(* IEC 61131-3 sources: horner-cscape-mcp/fixtures/st_library, 17 files *)

(* ---- analog_scaling_bounds.st ---- *)
(* ============================================================================
 * Title:       FB_AnalogScalingOutOfBounds
 * Description: Industrial Analog Scaling with Out-of-Bounds & Sensor Diagnostics.
 * Features:
 *   - Linear interpolation: Raw ADC / mA counts to Engineering Units (EU)
 *   - Out-of-bounds detection: 4-20mA open-loop wire-break and short-circuit faults
 *   - Configurable exponential smoothing digital filter for noisy plant signals
 *   - Output clamping to user process limits
 *   - Fail-safe fallback strategies (Hold Last Valid or Drive to Safe Preset)
 *   - Real-time sensor quality status and latched diagnostic error codes
 * Language:    IEC 61131-3 Structured Text (Pure ST)
 * ============================================================================ *)

FUNCTION_BLOCK FB_AnalogScalingOutOfBounds
VAR_INPUT
    RawIn : REAL := 0.0;                  (* Unscaled raw analog reading from ADC / PLC input *)
    RawMin : REAL := 4000.0;              (* Raw value corresponding to 0% range (e.g. 4.00 mA = 4000) *)
    RawMax : REAL := 20000.0;             (* Raw value corresponding to 100% range (e.g. 20.00 mA = 20000) *)
    EngMin : REAL := 0.0;                 (* Engineering units minimum (e.g. 0.0 Bar, Deg C, or RPM) *)
    EngMax : REAL := 100.0;               (* Engineering units maximum (e.g. 100.0 Bar, Deg C, or RPM) *)
    UnderflowTolerance : REAL := 400.0;   (* Margin below RawMin before declaring wire break (e.g. < 3.6 mA) *)
    OverflowTolerance : REAL := 800.0;    (* Margin above RawMax before declaring short circuit (e.g. > 20.8 mA) *)
    ClampOutput : BOOL := TRUE;           (* TRUE = constrain output between EngMin and EngMax *)
    FilterAlpha : REAL := 0.20;           (* Digital 1st-order filter factor (0.01 = heavy, 1.0 = bypass) *)
    FailSafeMode : INT := 0;              (* Fallback action on fault: 0 = Preset SafeValue, 1 = Hold Last Valid *)
    FailSafeValue : REAL := 0.0;          (* Fallback value emitted when FailSafeMode = 0 during fault *)
    ResetFault : BOOL := FALSE;           (* Pushbutton input to reset latched fault flags *)
END_VAR

VAR_OUTPUT
    ScaledValue : REAL := 0.0;            (* Final conditioned engineering units value *)
    RawFiltered : REAL := 0.0;            (* Filtered raw analog signal before scaling *)
    QualityOK : BOOL := TRUE;             (* Sensor signal is healthy and within legal electrical bounds *)
    AlarmUnderflow : BOOL := FALSE;       (* Active wire-break / open-loop / disconnected transmitter *)
    AlarmOverflow : BOOL := FALSE;        (* Active over-current / wiring short / ADC saturation *)
    LatchedFault : BOOL := FALSE;         (* Latch indicating an abnormal electrical event occurred *)
    ErrorCode : INT := 0;                 (* Diagnostics: 0=OK, 1=Underflow/Break, 2=Overflow/Short, 3=Config *)
END_VAR

VAR
    RawSpan : REAL := 16000.0;            (* Calculated raw range (RawMax - RawMin) *)
    EngSpan : REAL := 100.0;              (* Calculated engineering range (EngMax - EngMin) *)
    NormalizedFrac : REAL := 0.0;         (* Fraction between 0.0 and 1.0 *)
    CalculatedEng : REAL := 0.0;          (* Scaled value before clamping *)
    LastValidValue : REAL := 0.0;         (* Memory storing last known healthy measurement *)
    FilterInitialized : BOOL := FALSE;    (* Flag for initializing filter on first scan *)
END_VAR

(* 1. Reset Diagnostic Faults *)
IF ResetFault THEN
    LatchedFault := FALSE;
    ErrorCode := 0;
END_IF;

(* 2. Configuration Validation *)
RawSpan := RawMax - RawMin;
EngSpan := EngMax - EngMin;

IF ABS(RawSpan) < 0.001 THEN
    QualityOK := FALSE;
    LatchedFault := TRUE;
    ErrorCode := 3; (* Invalid configuration: zero raw span *)
    ScaledValue := FailSafeValue;
    RETURN;
END_IF;

(* 3. First-Order Digital Low-Pass Noise Filter *)
IF NOT FilterInitialized THEN
    RawFiltered := RawIn;
    FilterInitialized := TRUE;
ELSE
    RawFiltered := (FilterAlpha * RawIn) + ((1.0 - FilterAlpha) * RawFiltered);
END_IF;

(* 4. Out-of-Bounds Electrical Limit Verification *)
AlarmUnderflow := RawFiltered < (RawMin - UnderflowTolerance);
AlarmOverflow  := RawFiltered > (RawMax + OverflowTolerance);

IF AlarmUnderflow THEN
    QualityOK := FALSE;
    LatchedFault := TRUE;
    ErrorCode := 1; (* Wire break / open loop *)
ELSIF AlarmOverflow THEN
    QualityOK := FALSE;
    LatchedFault := TRUE;
    ErrorCode := 2; (* Over-range / short circuit *)
ELSE
    QualityOK := TRUE;
    IF NOT LatchedFault THEN
        ErrorCode := 0;
    END_IF;
END_IF;

(* 5. Scaling Calculation and Failsafe Strategy *)
IF QualityOK THEN
    (* Linear Scaling: EngMin + ((Raw - RawMin) / RawSpan) * EngSpan *)
    NormalizedFrac := (RawFiltered - RawMin) / RawSpan;
    CalculatedEng := EngMin + (NormalizedFrac * EngSpan);

    IF ClampOutput THEN
        IF EngMax >= EngMin THEN
            ScaledValue := LIMIT(EngMin, CalculatedEng, EngMax);
        ELSE
            ScaledValue := LIMIT(EngMax, CalculatedEng, EngMin);
        END_IF;
    ELSE
        ScaledValue := CalculatedEng;
    END_IF;

    LastValidValue := ScaledValue;
ELSE
    (* Sensor Fault: Apply Configured Failsafe Strategy *)
    IF FailSafeMode = 1 THEN
        ScaledValue := LastValidValue; (* Hold Last Valid *)
    ELSE
        ScaledValue := FailSafeValue;  (* Drive to Safe Preset *)
    END_IF;
END_IF;

END_FUNCTION_BLOCK

(* ---- condenser_hotwell_vacuum_control.st ---- *)
(* ============================================================================
 * Title:       FB_CondenserHotwellVacuumControl
 * Description: Turbine Surface Condenser Hotwell Level, Vacuum Deaeration &
 *              Circulating Water Cooling Tower Control.
 * IEC 61131-3: Pure Structured Text (ST) Only. Ladder logic strictly rejected.
 * OCS Mapping:
 *   %R125: Hotwell_Level_PV (tenths of inches: 0..1000, normal 500 = 50.0 in)
 *   %R126: Condenser_Vacuum_PV (hundredths of inHg abs: normal 150 = 1.50 inHg abs)
 *   %R127: Condensate_Dump_CV (0..100% dump valve to Condensate Storage Tank)
 *   %R128: Condensate_Makeup_CV (0..100% makeup valve from CST)
 *   %R129: Cooling_Tower_Basin_Temp_PV (tenths of deg F: normal 850 = 85.0 deg F)
 *   %R130: Cation_Conductivity_PV (hundredths of uS/cm: normal 20 = 0.20 uS/cm)
 *   %Q35:  Condensate_Pumps_Run (Digital output: Condensate extraction pumps)
 *   %Q36:  SJAE_Aux_Vacuum_Ejector (Digital output: Steam-jet air ejector / hogger)
 *   %Q37:  Cooling_Tower_Fan1 (Digital output: Stage 1 cooling fan)
 *   %Q38:  Cooling_Tower_Fan2 (Digital output: Stage 2 cooling fan)
 *   %Q39:  Condensate_Polisher_Bypass_Permit (Digital output: Polisher bypass)
 *   %M51:  Hotwell_Level_LowLow_Trip (Marker: Pump cavitation protection trip)
 *   %M52:  Condenser_Vacuum_HighHigh_Trip (Marker: Turbine backpressure trip)
 *   %M53:  Hotwell_Level_High_Alarm (Marker: Hotwell high level alarm)
 *   %M54:  Condenser_Tube_Leak_Alarm (Marker: Tube leak / cooling water ingress)
 * ============================================================================ *)

FUNCTION_BLOCK FB_CondenserHotwellVacuumControl
VAR_INPUT
    Hotwell_Level_PV : REAL := 500.0;            (* Tenths of inches (500.0 = 50.0 in) *)
    Condenser_Vacuum_PV : REAL := 150.0;         (* Hundredths inHg abs (150.0 = 1.50 inHg) *)
    Cooling_Tower_Basin_Temp_PV : REAL := 850.0; (* Tenths deg F (850.0 = 85.0 deg F) *)
    Cation_Conductivity_PV : REAL := 20.0;       (* Hundredths uS/cm (20.0 = 0.20 uS/cm) *)
    Permissive_Run : BOOL := TRUE;               (* Plant master permissive *)
    Reset_Alarms : BOOL := FALSE;                (* Operator alarm reset *)
END_VAR

VAR_OUTPUT
    Condensate_Dump_CV : REAL := 0.0;            (* 0.0 to 100.0 % *)
    Condensate_Makeup_CV : REAL := 0.0;          (* 0.0 to 100.0 % *)
    Condensate_Pumps_Run : BOOL := TRUE;
    SJAE_Aux_Vacuum_Ejector : BOOL := FALSE;
    Cooling_Tower_Fan1 : BOOL := FALSE;
    Cooling_Tower_Fan2 : BOOL := FALSE;
    Condensate_Polisher_Bypass_Permit : BOOL := TRUE;
    Hotwell_Level_LowLow_Trip : BOOL := FALSE;
    Condenser_Vacuum_HighHigh_Trip : BOOL := FALSE;
    Hotwell_Level_High_Alarm : BOOL := FALSE;
    Condenser_Tube_Leak_Alarm : BOOL := FALSE;
END_VAR

VAR
    Level_Error : REAL := 0.0;
END_VAR

(* Reset Latches if requested *)
IF Reset_Alarms THEN
    Hotwell_Level_LowLow_Trip := FALSE;
    Condenser_Vacuum_HighHigh_Trip := FALSE;
    Hotwell_Level_High_Alarm := FALSE;
    Condenser_Tube_Leak_Alarm := FALSE;
END_IF;

(* 1. Hotwell Level Control & Cavitation Protection *)
IF Hotwell_Level_PV <= 100.0 THEN
    (* Low-Low Level: Trip Condensate Extraction Pumps immediately *)
    Hotwell_Level_LowLow_Trip := TRUE;
    Condensate_Pumps_Run := FALSE;
    Condensate_Makeup_CV := 100.0;
    Condensate_Dump_CV := 0.0;
ELSIF Hotwell_Level_PV >= 750.0 THEN
    (* High Level: Open Dump Valve to CST, Inhibit Makeup *)
    Hotwell_Level_High_Alarm := TRUE;
    Condensate_Dump_CV := (Hotwell_Level_PV - 750.0) * 0.4;
    IF Condensate_Dump_CV > 100.0 THEN
        Condensate_Dump_CV := 100.0;
    END_IF;
    Condensate_Makeup_CV := 0.0;
    IF Permissive_Run AND NOT Hotwell_Level_LowLow_Trip THEN
        Condensate_Pumps_Run := TRUE;
    END_IF;
ELSIF Hotwell_Level_PV <= 300.0 THEN
    (* Low Level: Open Makeup Valve from CST, Close Dump *)
    Condensate_Makeup_CV := (300.0 - Hotwell_Level_PV) * 0.5;
    IF Condensate_Makeup_CV > 100.0 THEN
        Condensate_Makeup_CV := 100.0;
    END_IF;
    Condensate_Dump_CV := 0.0;
    IF Permissive_Run AND NOT Hotwell_Level_LowLow_Trip THEN
        Condensate_Pumps_Run := TRUE;
    END_IF;
ELSE
    (* Normal Hotwell Equilibrium *)
    Condensate_Dump_CV := 0.0;
    Condensate_Makeup_CV := 0.0;
    Hotwell_Level_High_Alarm := FALSE;
    IF Permissive_Run AND NOT Hotwell_Level_LowLow_Trip THEN
        Condensate_Pumps_Run := TRUE;
    END_IF;
END_IF;

(* 2. Condenser Vacuum & Air Ejection Control *)
IF Condenser_Vacuum_PV >= 500.0 THEN
    (* Vacuum Loss High-High Trip (5.0 inHg abs) *)
    Condenser_Vacuum_HighHigh_Trip := TRUE;
    SJAE_Aux_Vacuum_Ejector := TRUE;
ELSIF Condenser_Vacuum_PV >= 350.0 THEN
    (* Vacuum Deteriorating: Engage Auxiliary Air Ejector / Hogger *)
    SJAE_Aux_Vacuum_Ejector := TRUE;
ELSE
    (* Normal Vacuum (<= 3.50 inHg abs) *)
    SJAE_Aux_Vacuum_Ejector := FALSE;
END_IF;

(* 3. Circulating Water Cooling Tower Fan Staging *)
IF Cooling_Tower_Basin_Temp_PV >= 980.0 THEN
    (* High Temp: Stage 1 and Stage 2 Fans Running *)
    Cooling_Tower_Fan1 := TRUE;
    Cooling_Tower_Fan2 := TRUE;
ELSIF Cooling_Tower_Basin_Temp_PV >= 920.0 THEN
    (* Moderate Temp: Stage 1 Fan Running *)
    Cooling_Tower_Fan1 := TRUE;
    Cooling_Tower_Fan2 := FALSE;
ELSE
    (* Normal / Cool Basin Temp *)
    Cooling_Tower_Fan1 := FALSE;
    Cooling_Tower_Fan2 := FALSE;
END_IF;

(* 4. Tube Leak / Raw Cooling Water Ingress Detection *)
IF Cation_Conductivity_PV >= 200.0 THEN
    (* Water Ingress Alert: Trip Polisher Bypass, Latch Alarm *)
    Condenser_Tube_Leak_Alarm := TRUE;
    Condensate_Polisher_Bypass_Permit := FALSE;
ELSE
    Condensate_Polisher_Bypass_Permit := TRUE;
END_IF;

END_FUNCTION_BLOCK

(* ---- conveyor_sorting_state_machine.st ---- *)
(* ============================================================================
 * Title:       FB_ConveyorSortingStateMachine
 * Description: High-Speed Material Handling Conveyor Sortation State Machine.
 * Features:
 *   - Structured CASE-based state machine for packaging & sortation lines
 *   - Debounced optical presence sensing at infeed
 *   - Barcode classification routing to Lane 1, Lane 2, or Reject Chute
 *   - Pneumatic diverter actuation with cylinder end-switch verification
 *   - Jam detection timer with automatic reverse jog clearing routine
 *   - Hardware emergency-stop and line stop supervisory interlocks
 *   - Real-time production piece counters (Total, Lanes, Rejects)
 * Language:    IEC 61131-3 Structured Text (Pure ST)
 * ============================================================================ *)

FUNCTION_BLOCK FB_ConveyorSortingStateMachine
VAR_INPUT
    Enable : BOOL := TRUE;                (* Master system run permissive *)
    StartPB : BOOL := FALSE;              (* System start push button *)
    StopPB : BOOL := FALSE;               (* System normal stop push button *)
    EStop : BOOL := TRUE;                 (* Emergency stop circuit (TRUE = Normal/Healthy) *)
    PackageDetectPE : BOOL := FALSE;      (* Optical sensor detecting parcel at inspection point *)
    BarcodeScanValid : BOOL := FALSE;     (* Strobe from vision / barcode reader when decode ready *)
    BarcodeDestLane : INT := 1;           (* Target destination from scanner: 1=Lane1, 2=Lane2, 3=Reject *)
    Diverter1_Extended : BOOL := FALSE;   (* Reed switch: Diverter 1 fully extended *)
    Diverter2_Extended : BOOL := FALSE;   (* Reed switch: Diverter 2 fully extended *)
    DivertersRetracted : BOOL := TRUE;    (* Reed switches: Both diverters back in home position *)
    ExitPE_Lane1 : BOOL := FALSE;         (* Optical sensor at Lane 1 discharge *)
    ExitPE_Lane2 : BOOL := FALSE;         (* Optical sensor at Lane 2 discharge *)
    ExitPE_Reject : BOOL := FALSE;        (* Optical sensor at Reject chute discharge *)
    ResetFault : BOOL := FALSE;           (* Push button to clear latched faults *)
    JamTimeoutSec : REAL := 4.0;          (* Maximum transit time before declaring parcel jam *)
    DivertStrokeSec : REAL := 1.2;        (* Cylinder stroke timeout limit (seconds) *)
    CycleTimeSec : REAL := 0.1;           (* Scan cycle delta time (seconds) *)
END_VAR

VAR_OUTPUT
    ConveyorRun : BOOL := FALSE;          (* Motor contactor / VFD forward command *)
    ConveyorRev : BOOL := FALSE;          (* Motor contactor / VFD reverse command for clearing *)
    Diverter1_Extend : BOOL := FALSE;     (* Pneumatic cylinder solenoid for Lane 1 *)
    Diverter2_Extend : BOOL := FALSE;     (* Pneumatic cylinder solenoid for Lane 2 *)
    RejectGate_Extend : BOOL := FALSE;    (* Pneumatic cylinder solenoid for Reject chute *)
    CurrentState : INT := 0;              (* Numeric state code for HMI diagnostics *)
    JamAlarm : BOOL := FALSE;             (* Latched conveyor jam condition *)
    DiverterFault : BOOL := FALSE;        (* Diverter cylinder failure to extend/retract *)
    CountTotal : DINT := 0;               (* Total parcels successfully processed *)
    CountLane1 : DINT := 0;               (* Total parcels diverted to Lane 1 *)
    CountLane2 : DINT := 0;               (* Total parcels diverted to Lane 2 *)
    CountReject : DINT := 0;              (* Total parcels diverted to Reject *)
END_VAR

VAR
    StateTimer : REAL := 0.0;             (* Dwell timer in active state *)
    JamTimer : REAL := 0.0;               (* Accumulator for parcel transit watchdog *)
    InfeedDebounce : REAL := 0.0;         (* Infeed optical filter accumulator *)
    InfeedConfirmed : BOOL := FALSE;      (* Debounced parcel detection flag *)
    LatchedLane : INT := 1;               (* Stored destination for current parcel *)
    RunPermissive : BOOL := FALSE;        (* Running latch set by StartPB, cleared by StopPB *)
END_VAR

(* 1. Safety and Fault Management *)
IF ResetFault THEN
    JamAlarm := FALSE;
    DiverterFault := FALSE;
END_IF;

IF NOT EStop THEN
    CurrentState := 99; (* Emergency Stop *)
    RunPermissive := FALSE;
ELSIF StopPB THEN
    RunPermissive := FALSE;
ELSIF StartPB AND Enable AND (NOT JamAlarm) AND (NOT DiverterFault) THEN
    RunPermissive := TRUE;
END_IF;

IF JamAlarm OR DiverterFault THEN
    RunPermissive := FALSE;
END_IF;

(* 2. Optical Sensor Debounce (50 ms noise immunity) *)
IF PackageDetectPE THEN
    InfeedDebounce := InfeedDebounce + CycleTimeSec;
    IF InfeedDebounce >= 0.05 THEN
        InfeedConfirmed := TRUE;
    END_IF;
ELSE
    InfeedDebounce := 0.0;
    InfeedConfirmed := FALSE;
END_IF;

(* 3. State Machine Execution *)
CASE CurrentState OF

    0: (* STATE_IDLE: Waiting for line start permissive *)
        ConveyorRun := FALSE;
        ConveyorRev := FALSE;
        Diverter1_Extend := FALSE;
        Diverter2_Extend := FALSE;
        RejectGate_Extend := FALSE;
        StateTimer := 0.0;
        JamTimer := 0.0;

        IF RunPermissive AND DivertersRetracted THEN
            CurrentState := 10;
        END_IF;

    10: (* STATE_FEED: Conveyor running, awaiting package arrival *)
        ConveyorRun := TRUE;
        ConveyorRev := FALSE;
        Diverter1_Extend := FALSE;
        Diverter2_Extend := FALSE;
        RejectGate_Extend := FALSE;

        IF NOT RunPermissive THEN
            CurrentState := 0;
        ELSIF InfeedConfirmed THEN
            StateTimer := 0.0;
            CurrentState := 20;
        END_IF;

    20: (* STATE_INSPECT: Package present, acquiring barcode/classification *)
        ConveyorRun := TRUE;
        StateTimer := StateTimer + CycleTimeSec;

        IF BarcodeScanValid THEN
            LatchedLane := BarcodeDestLane;
            StateTimer := 0.0;
            JamTimer := 0.0;
            IF LatchedLane = 1 THEN
                CurrentState := 30;
            ELSIF LatchedLane = 2 THEN
                CurrentState := 40;
            ELSE
                CurrentState := 50;
            END_IF;
        ELSIF StateTimer >= 1.5 THEN
            (* Scanner timeout: Default route to Reject *)
            LatchedLane := 3;
            StateTimer := 0.0;
            JamTimer := 0.0;
            CurrentState := 50;
        END_IF;

    30: (* STATE_DIVERT_LANE1: Actuate Diverter 1 *)
        ConveyorRun := TRUE;
        Diverter1_Extend := TRUE;
        StateTimer := StateTimer + CycleTimeSec;
        JamTimer := JamTimer + CycleTimeSec;

        (* Check end switch feedback *)
        IF StateTimer >= DivertStrokeSec AND (NOT Diverter1_Extended) THEN
            DiverterFault := TRUE;
            CurrentState := 90;
        ELSIF ExitPE_Lane1 OR (StateTimer >= 2.5) THEN
            (* Package diverted successfully *)
            CountLane1 := CountLane1 + 1;
            CountTotal := CountTotal + 1;
            Diverter1_Extend := FALSE;
            CurrentState := 60;
        ELSIF JamTimer >= JamTimeoutSec THEN
            JamAlarm := TRUE;
            CurrentState := 90;
        END_IF;

    40: (* STATE_DIVERT_LANE2: Actuate Diverter 2 *)
        ConveyorRun := TRUE;
        Diverter2_Extend := TRUE;
        StateTimer := StateTimer + CycleTimeSec;
        JamTimer := JamTimer + CycleTimeSec;

        IF StateTimer >= DivertStrokeSec AND (NOT Diverter2_Extended) THEN
            DiverterFault := TRUE;
            CurrentState := 90;
        ELSIF ExitPE_Lane2 OR (StateTimer >= 2.5) THEN
            CountLane2 := CountLane2 + 1;
            CountTotal := CountTotal + 1;
            Diverter2_Extend := FALSE;
            CurrentState := 60;
        ELSIF JamTimer >= JamTimeoutSec THEN
            JamAlarm := TRUE;
            CurrentState := 90;
        END_IF;

    50: (* STATE_REJECT: Actuate Reject gate / Chute *)
        ConveyorRun := TRUE;
        RejectGate_Extend := TRUE;
        StateTimer := StateTimer + CycleTimeSec;
        JamTimer := JamTimer + CycleTimeSec;

        IF ExitPE_Reject OR (StateTimer >= 2.5) THEN
            CountReject := CountReject + 1;
            CountTotal := CountTotal + 1;
            RejectGate_Extend := FALSE;
            CurrentState := 60;
        ELSIF JamTimer >= JamTimeoutSec THEN
            JamAlarm := TRUE;
            CurrentState := 90;
        END_IF;

    60: (* STATE_PACKAGE_CLEARED: Ensure actuators home before next item *)
        ConveyorRun := TRUE;
        Diverter1_Extend := FALSE;
        Diverter2_Extend := FALSE;
        RejectGate_Extend := FALSE;
        StateTimer := StateTimer + CycleTimeSec;

        IF DivertersRetracted AND (NOT InfeedConfirmed) THEN
            IF RunPermissive THEN
                CurrentState := 10;
            ELSE
                CurrentState := 0;
            END_IF;
        ELSIF StateTimer >= 3.0 THEN
            (* Actuators stuck in lane *)
            DiverterFault := TRUE;
            CurrentState := 90;
        END_IF;

    90: (* STATE_JAM_FAULT: Line halted on jam or cylinder failure *)
        ConveyorRun := FALSE;
        ConveyorRev := FALSE;
        Diverter1_Extend := FALSE;
        Diverter2_Extend := FALSE;
        RejectGate_Extend := FALSE;

        IF (NOT JamAlarm) AND (NOT DiverterFault) AND DivertersRetracted THEN
            CurrentState := 0;
        END_IF;

    99: (* STATE_ESTOP: Emergency Stop engaged *)
        ConveyorRun := FALSE;
        ConveyorRev := FALSE;
        Diverter1_Extend := FALSE;
        Diverter2_Extend := FALSE;
        RejectGate_Extend := FALSE;

        IF EStop AND (NOT RunPermissive) THEN
            CurrentState := 0;
        END_IF;

    ELSE
        CurrentState := 0;
END_CASE;

END_FUNCTION_BLOCK

(* ---- first_fault_annunciator.st ---- *)
(* ============================================================================
 * Title:       FB_FirstFaultAnnunciator
 * Description: ISA-18.2 8-Point First-Out Alarm Annunciator with Visual & Audio Logic.
 * Features:
 *   - First-out discrimination: Identifies root-cause trip in cascading outages
 *   - Visual flashing states: Fast flash (First-Out), Slow flash (Subsequent)
 *   - Steady illumination upon operator acknowledgment
 *   - Audible horn driving with silence/acknowledge push button
 *   - Reset interlock: Alarms clear only when field conditions return to normal
 *   - Lamp Test pushbutton to verify panel indicators and audible sounder
 * Language:    IEC 61131-3 Structured Text (Pure ST)
 * ============================================================================ *)

FUNCTION_BLOCK FB_FirstFaultAnnunciator
VAR_INPUT
    AlarmIn1 : BOOL := FALSE;             (* Point 1: e.g. Emergency Stop tripped *)
    AlarmIn2 : BOOL := FALSE;             (* Point 2: e.g. High-High Vessel Pressure *)
    AlarmIn3 : BOOL := FALSE;             (* Point 3: e.g. High-High Reactor Temperature *)
    AlarmIn4 : BOOL := FALSE;             (* Point 4: e.g. Low-Low Lube Oil Pressure *)
    AlarmIn5 : BOOL := FALSE;             (* Point 5: e.g. Motor Overload Breaker *)
    AlarmIn6 : BOOL := FALSE;             (* Point 6: e.g. Sump High Spill Level *)
    AlarmIn7 : BOOL := FALSE;             (* Point 7: e.g. Instrument Air Low Pressure *)
    AlarmIn8 : BOOL := FALSE;             (* Point 8: e.g. Combustible Gas Detector *)
    AckPB : BOOL := FALSE;                (* Operator Acknowledge push button *)
    ResetPB : BOOL := FALSE;              (* Operator Reset push button *)
    TestPB : BOOL := FALSE;               (* Lamp / Horn Test push button *)
    CycleTimeSec : REAL := 0.1;           (* Scan delta time (seconds) *)
END_VAR

VAR_OUTPUT
    Horn : BOOL := FALSE;                 (* Digital output: Audible alarm sounder *)
    Beacon1 : BOOL := FALSE;              (* Digital output: Lamp for Point 1 *)
    Beacon2 : BOOL := FALSE;              (* Digital output: Lamp for Point 2 *)
    Beacon3 : BOOL := FALSE;              (* Digital output: Lamp for Point 3 *)
    Beacon4 : BOOL := FALSE;              (* Digital output: Lamp for Point 4 *)
    Beacon5 : BOOL := FALSE;              (* Digital output: Lamp for Point 5 *)
    Beacon6 : BOOL := FALSE;              (* Digital output: Lamp for Point 6 *)
    Beacon7 : BOOL := FALSE;              (* Digital output: Lamp for Point 7 *)
    Beacon8 : BOOL := FALSE;              (* Digital output: Lamp for Point 8 *)
    FirstOutId : INT := 0;                (* ID of the root-cause first alarm (1 to 8, 0=None) *)
    AnyAlarmActive : BOOL := FALSE;       (* TRUE if any alarm is currently in alarm state *)
    AnyUnack : BOOL := FALSE;             (* TRUE if any alarm remains unacknowledged *)
END_VAR

VAR
    FlashTimerFast : REAL := 0.0;         (* Accumulator for 2.0 Hz fast flasher *)
    FlashTimerSlow : REAL := 0.0;         (* Accumulator for 1.0 Hz slow flasher *)
    FlashFastState : BOOL := FALSE;       (* Fast flash toggle signal *)
    FlashSlowState : BOOL := FALSE;       (* Slow flash toggle signal *)
    Latched1 : BOOL := FALSE;             (* Latched alarm state for Point 1 *)
    Latched2 : BOOL := FALSE;             (* Latched alarm state for Point 2 *)
    Latched3 : BOOL := FALSE;             (* Latched alarm state for Point 3 *)
    Latched4 : BOOL := FALSE;             (* Latched alarm state for Point 4 *)
    Latched5 : BOOL := FALSE;             (* Latched alarm state for Point 5 *)
    Latched6 : BOOL := FALSE;             (* Latched alarm state for Point 6 *)
    Latched7 : BOOL := FALSE;             (* Latched alarm state for Point 7 *)
    Latched8 : BOOL := FALSE;             (* Latched alarm state for Point 8 *)
    Ack1 : BOOL := FALSE;                 (* Acknowledged state for Point 1 *)
    Ack2 : BOOL := FALSE;                 (* Acknowledged state for Point 2 *)
    Ack3 : BOOL := FALSE;                 (* Acknowledged state for Point 3 *)
    Ack4 : BOOL := FALSE;                 (* Acknowledged state for Point 4 *)
    Ack5 : BOOL := FALSE;                 (* Acknowledged state for Point 5 *)
    Ack6 : BOOL := FALSE;                 (* Acknowledged state for Point 6 *)
    Ack7 : BOOL := FALSE;                 (* Acknowledged state for Point 7 *)
    Ack8 : BOOL := FALSE;                 (* Acknowledged state for Point 8 *)
END_VAR

(* 1. Flasher Oscillators (Fast = 250ms half-period, Slow = 500ms half-period) *)
FlashTimerFast := FlashTimerFast + CycleTimeSec;
IF FlashTimerFast >= 0.25 THEN
    FlashTimerFast := 0.0;
    FlashFastState := NOT FlashFastState;
END_IF;

FlashTimerSlow := FlashTimerSlow + CycleTimeSec;
IF FlashTimerSlow >= 0.50 THEN
    FlashTimerSlow := 0.0;
    FlashSlowState := NOT FlashSlowState;
END_IF;

(* 2. First-Out Latching and Point Alarm Acquisition *)
IF AlarmIn1 THEN Latched1 := TRUE; END_IF;
IF AlarmIn2 THEN Latched2 := TRUE; END_IF;
IF AlarmIn3 THEN Latched3 := TRUE; END_IF;
IF AlarmIn4 THEN Latched4 := TRUE; END_IF;
IF AlarmIn5 THEN Latched5 := TRUE; END_IF;
IF AlarmIn6 THEN Latched6 := TRUE; END_IF;
IF AlarmIn7 THEN Latched7 := TRUE; END_IF;
IF AlarmIn8 THEN Latched8 := TRUE; END_IF;

IF FirstOutId = 0 THEN
    IF AlarmIn1 THEN FirstOutId := 1;
    ELSIF AlarmIn2 THEN FirstOutId := 2;
    ELSIF AlarmIn3 THEN FirstOutId := 3;
    ELSIF AlarmIn4 THEN FirstOutId := 4;
    ELSIF AlarmIn5 THEN FirstOutId := 5;
    ELSIF AlarmIn6 THEN FirstOutId := 6;
    ELSIF AlarmIn7 THEN FirstOutId := 7;
    ELSIF AlarmIn8 THEN FirstOutId := 8;
    END_IF;
END_IF;

(* 3. Operator Acknowledge PB *)
IF AckPB THEN
    IF Latched1 THEN Ack1 := TRUE; END_IF;
    IF Latched2 THEN Ack2 := TRUE; END_IF;
    IF Latched3 THEN Ack3 := TRUE; END_IF;
    IF Latched4 THEN Ack4 := TRUE; END_IF;
    IF Latched5 THEN Ack5 := TRUE; END_IF;
    IF Latched6 THEN Ack6 := TRUE; END_IF;
    IF Latched7 THEN Ack7 := TRUE; END_IF;
    IF Latched8 THEN Ack8 := TRUE; END_IF;
END_IF;

(* 4. Operator Reset PB (clears points only if field sensor is normal AND acknowledged) *)
IF ResetPB THEN
    IF Ack1 AND (NOT AlarmIn1) THEN Latched1 := FALSE; Ack1 := FALSE; END_IF;
    IF Ack2 AND (NOT AlarmIn2) THEN Latched2 := FALSE; Ack2 := FALSE; END_IF;
    IF Ack3 AND (NOT AlarmIn3) THEN Latched3 := FALSE; Ack3 := FALSE; END_IF;
    IF Ack4 AND (NOT AlarmIn4) THEN Latched4 := FALSE; Ack4 := FALSE; END_IF;
    IF Ack5 AND (NOT AlarmIn5) THEN Latched5 := FALSE; Ack5 := FALSE; END_IF;
    IF Ack6 AND (NOT AlarmIn6) THEN Latched6 := FALSE; Ack6 := FALSE; END_IF;
    IF Ack7 AND (NOT AlarmIn7) THEN Latched7 := FALSE; Ack7 := FALSE; END_IF;
    IF Ack8 AND (NOT AlarmIn8) THEN Latched8 := FALSE; Ack8 := FALSE; END_IF;

    (* Reset FirstOutId if all latches have cleared *)
    IF (NOT Latched1) AND (NOT Latched2) AND (NOT Latched3) AND (NOT Latched4) AND (NOT Latched5) AND (NOT Latched6) AND (NOT Latched7) AND (NOT Latched8) THEN
        FirstOutId := 0;
    END_IF;
END_IF;

(* 5. Supervisory Summary Flags *)
AnyAlarmActive := Latched1 OR Latched2 OR Latched3 OR Latched4 OR Latched5 OR Latched6 OR Latched7 OR Latched8;

AnyUnack := (Latched1 AND NOT Ack1) OR (Latched2 AND NOT Ack2) OR (Latched3 AND NOT Ack3) OR (Latched4 AND NOT Ack4) OR (Latched5 AND NOT Ack5) OR (Latched6 AND NOT Ack6) OR (Latched7 AND NOT Ack7) OR (Latched8 AND NOT Ack8);

(* 6. Audible Horn Logic *)
IF TestPB THEN
    Horn := TRUE;
ELSIF AnyUnack THEN
    Horn := TRUE;
ELSE
    Horn := FALSE;
END_IF;

(* 7. Visual Beacon Illumination Logic *)
IF TestPB THEN
    Beacon1 := TRUE; Beacon2 := TRUE; Beacon3 := TRUE; Beacon4 := TRUE;
    Beacon5 := TRUE; Beacon6 := TRUE; Beacon7 := TRUE; Beacon8 := TRUE;
ELSE
    (* Point 1 *)
    IF NOT Latched1 THEN Beacon1 := FALSE;
    ELSIF FirstOutId = 1 AND (NOT Ack1) THEN Beacon1 := FlashFastState;
    ELSIF NOT Ack1 THEN Beacon1 := FlashSlowState;
    ELSE Beacon1 := TRUE;
    END_IF;

    (* Point 2 *)
    IF NOT Latched2 THEN Beacon2 := FALSE;
    ELSIF FirstOutId = 2 AND (NOT Ack2) THEN Beacon2 := FlashFastState;
    ELSIF NOT Ack2 THEN Beacon2 := FlashSlowState;
    ELSE Beacon2 := TRUE;
    END_IF;

    (* Point 3 *)
    IF NOT Latched3 THEN Beacon3 := FALSE;
    ELSIF FirstOutId = 3 AND (NOT Ack3) THEN Beacon3 := FlashFastState;
    ELSIF NOT Ack3 THEN Beacon3 := FlashSlowState;
    ELSE Beacon3 := TRUE;
    END_IF;

    (* Point 4 *)
    IF NOT Latched4 THEN Beacon4 := FALSE;
    ELSIF FirstOutId = 4 AND (NOT Ack4) THEN Beacon4 := FlashFastState;
    ELSIF NOT Ack4 THEN Beacon4 := FlashSlowState;
    ELSE Beacon4 := TRUE;
    END_IF;

    (* Point 5 *)
    IF NOT Latched5 THEN Beacon5 := FALSE;
    ELSIF FirstOutId = 5 AND (NOT Ack5) THEN Beacon5 := FlashFastState;
    ELSIF NOT Ack5 THEN Beacon5 := FlashSlowState;
    ELSE Beacon5 := TRUE;
    END_IF;

    (* Point 6 *)
    IF NOT Latched6 THEN Beacon6 := FALSE;
    ELSIF FirstOutId = 6 AND (NOT Ack6) THEN Beacon6 := FlashFastState;
    ELSIF NOT Ack6 THEN Beacon6 := FlashSlowState;
    ELSE Beacon6 := TRUE;
    END_IF;

    (* Point 7 *)
    IF NOT Latched7 THEN Beacon7 := FALSE;
    ELSIF FirstOutId = 7 AND (NOT Ack7) THEN Beacon7 := FlashFastState;
    ELSIF NOT Ack7 THEN Beacon7 := FlashSlowState;
    ELSE Beacon7 := TRUE;
    END_IF;

    (* Point 8 *)
    IF NOT Latched8 THEN Beacon8 := FALSE;
    ELSIF FirstOutId = 8 AND (NOT Ack8) THEN Beacon8 := FlashFastState;
    ELSIF NOT Ack8 THEN Beacon8 := FlashSlowState;
    ELSE Beacon8 := TRUE;
    END_IF;
END_IF;

END_FUNCTION_BLOCK

(* ---- flow_totalizer_integrator.st ---- *)
(* ============================================================================
 * Title:       FB_FlowTotalizer
 * Description: Industrial Fluid Flow Numerical Integrator & Telemetry Pulse Generator.
 * Features:
 *   - Trapezoidal numerical integration of instant flow rates to total volume
 *   - Low-flow cutoff threshold preventing measurement drift at near-zero flow
 *   - Triple accumulation tiers: Master Total, Daily Total, and Batch Total
 *   - Telemetry pulse generation: Fixed duration pulses for every N volume units
 *   - Forward and reverse flow direction qualification
 * Language:    IEC 61131-3 Structured Text (Pure ST)
 * ============================================================================ *)

FUNCTION_BLOCK FB_FlowTotalizer
VAR_INPUT
    FlowRate : REAL := 0.0;               (* Instantaneous fluid flow rate (e.g. m3/h, GPM, L/min) *)
    TimeBaseSec : REAL := 3600.0;         (* Time unit of flow rate in seconds (3600.0=hr, 60.0=min, 1.0=sec) *)
    LowFlowCutoff : REAL := 0.5;          (* Low flow threshold below which rate is forced to 0.0 *)
    ResetBatch : BOOL := FALSE;           (* Reset command for Batch Totalizer *)
    ResetDaily : BOOL := FALSE;           (* Reset command for Daily Totalizer *)
    ResetMaster : BOOL := FALSE;          (* Protected reset command for Master Totalizer *)
    PulseVolume : REAL := 10.0;           (* Volume units per telemetry pulse (e.g. 10.0 Liters) *)
    PulseDurationSec : REAL := 0.2;       (* Duration of each digital output pulse (seconds) *)
    CycleTimeSec : REAL := 0.1;           (* Execution scan period (seconds) *)
END_VAR

VAR_OUTPUT
    TotalMaster : LREAL := 0.0;           (* High-precision Master Total accumulated volume *)
    TotalDaily : REAL := 0.0;             (* Daily Resettable Total accumulated volume *)
    TotalBatch : REAL := 0.0;             (* Batch / Job Resettable Total volume *)
    NetFlowRate : REAL := 0.0;            (* Flow rate after low-flow cutoff qualification *)
    PulseOut : BOOL := FALSE;             (* Digital output pulse for remote telemetry / RTU *)
    PulseCount : DINT := 0;               (* Total number of volume pulses generated *)
END_VAR

VAR
    PrevRate : REAL := 0.0;               (* Previous scan flow rate for trapezoidal integration *)
    IncrementalVol : REAL := 0.0;         (* Volume accumulated during current scan cycle *)
    PulseVolumeAcc : REAL := 0.0;         (* Sub-pulse volume accumulator *)
    PulseTimer : REAL := 0.0;             (* Active pulse duration timer *)
END_VAR

(* 1. Manual and Automated Totalizer Resets *)
IF ResetMaster THEN
    TotalMaster := 0.0;
END_IF;

IF ResetDaily THEN
    TotalDaily := 0.0;
END_IF;

IF ResetBatch THEN
    TotalBatch := 0.0;
END_IF;

(* 2. Low-Flow Cutoff Evaluation *)
IF ABS(FlowRate) < LowFlowCutoff THEN
    NetFlowRate := 0.0;
ELSE
    NetFlowRate := FlowRate;
END_IF;

(* 3. Trapezoidal Numerical Integration: V = ((R1 + R0) / 2) * (dt / TimeBase) *)
IF TimeBaseSec > 0.001 THEN
    IncrementalVol := ((NetFlowRate + PrevRate) * 0.5) * (CycleTimeSec / TimeBaseSec);
ELSE
    IncrementalVol := 0.0;
END_IF;
PrevRate := NetFlowRate;

(* 4. Volume Accumulation Across Tiers *)
TotalMaster := TotalMaster + IncrementalVol;
TotalDaily := TotalDaily + IncrementalVol;
TotalBatch := TotalBatch + IncrementalVol;

(* 5. Telemetry Pulse Train Generation *)
IF PulseVolume > 0.001 THEN
    PulseVolumeAcc := PulseVolumeAcc + IncrementalVol;

    (* Trigger pulse when accumulated volume meets pulse threshold *)
    IF PulseVolumeAcc >= PulseVolume AND (NOT PulseOut) THEN
        PulseVolumeAcc := PulseVolumeAcc - PulseVolume;
        PulseOut := TRUE;
        PulseTimer := 0.0;
        PulseCount := PulseCount + 1;
    END_IF;

    (* Maintain pulse width for configured duration *)
    IF PulseOut THEN
        PulseTimer := PulseTimer + CycleTimeSec;
        IF PulseTimer >= PulseDurationSec THEN
            PulseOut := FALSE;
            PulseTimer := 0.0;
        END_IF;
    END_IF;
ELSE
    PulseOut := FALSE;
    PulseTimer := 0.0;
END_IF;

END_FUNCTION_BLOCK

(* ---- generator_avr_excitation_control.st ---- *)
(* ============================================================================
 * Title:       FB_GeneratorAvrExcitationControl
 * Description: Synchronous Generator Excitation & Automatic Voltage Regulator (AVR),
 *              Under-Excitation Limiter (UEL), Over-Excitation Limiter (OEL),
 *              Volts-Per-Hertz (V/Hz) Overfluxing & Loss-of-Field (40) Trip Interlock.
 * IEC 61131-3: Pure Structured Text (ST) Only. Ladder logic strictly rejected.
 * OCS Mapping:
 *   %R137: Generator_Terminal_Voltage_kV (INT: tenths of kV, e.g. 138 = 13.8 kV)
 *   %R138: Generator_Reactive_Power_MVAR (INT: tenths of MVAR, e.g. 150 = 15.0 MVAR)
 *   %R139: Excitation_Field_Current_Amps (INT: tenths of Amps, e.g. 420 = 42.0 A)
 *   %R140: Excitation_Field_Voltage_Volts (INT: Volts DC, e.g. 125 VDC)
 *   %R141: Grid_Bus_Voltage_kV (INT: tenths of kV, e.g. 138 = 13.8 kV)
 *   %R142: Generator_Frequency_Hz (INT: hundredths of Hz, e.g. 6000 = 60.00 Hz)
 *   %Q44:  AVR_Automatic_Mode_Active (BOOL: True = Auto AVR, False = Manual FCR)
 *   %Q45:  Field_Breaker_Close_Command (BOOL: Field contactor/breaker permit)
 *   %Q46:  Under_Excitation_Limiter_Active (BOOL: UEL active)
 *   %Q47:  Over_Excitation_Limiter_Active (BOOL: OEL active)
 *   %M58:  Volts_Per_Hertz_Overfluxing_Trip (BOOL: V/Hz overfluxing trip)
 *   %M59:  Generator_Loss_of_Field_Trip (BOOL: 40 relay loss of field trip)
 *   %M60:  Field_Overcurrent_Trip_Latched (BOOL: Latched field overcurrent)
 * ============================================================================ *)

FUNCTION_BLOCK FB_GeneratorAvrExcitationControl
VAR_INPUT
    Generator_Terminal_Voltage_kV : INT := 138;   (* Tenths kV (138 = 13.8 kV) *)
    Generator_Reactive_Power_MVAR : INT := 150;   (* Tenths MVAR (150 = 15.0 MVAR lag) *)
    Excitation_Field_Current_Amps : INT := 420;   (* Tenths A (420 = 42.0 A) *)
    Grid_Bus_Voltage_kV : INT := 138;             (* Tenths kV (138 = 13.8 kV) *)
    Generator_Frequency_Hz : INT := 6000;         (* Hundredths Hz (6000 = 60.00 Hz) *)
    AVR_Auto_Select : BOOL := TRUE;               (* Auto / Manual selector *)
    Master_Trip_Reset : BOOL := FALSE;            (* Trip reset PB *)
    Generator_Breaker_Closed : BOOL := TRUE;      (* Main generator breaker *)
END_VAR

VAR_OUTPUT
    AVR_Automatic_Mode_Active : BOOL := TRUE;
    Field_Breaker_Close_Command : BOOL := TRUE;
    Under_Excitation_Limiter_Active : BOOL := FALSE;
    Over_Excitation_Limiter_Active : BOOL := FALSE;
    Excitation_Field_Voltage_Volts : INT := 125;  (* Field VDC *)
    Volts_Per_Hertz_Overfluxing_Trip : BOOL := FALSE;
    Generator_Loss_of_Field_Trip : BOOL := FALSE;
    Field_Overcurrent_Trip_Latched : BOOL := FALSE;
END_VAR

VAR
    Rated_Voltage_kV : INT := 138;
    OEL_Threshold_Amps : INT := 700;              (* 70.0 A ceiling *)
    UEL_Threshold_MVAR : INT := -100;             (* -10.0 MVAR leading clamp *)
    Loss_of_Field_Threshold_MVAR : INT := -200;   (* -20.0 MVAR leading trip *)
    V_Per_Hz_Limit_Ratio : INT := 110;            (* 110% V/Hz *)
END_VAR

(* 0. Master Trip Reset *)
IF Master_Trip_Reset THEN
    Volts_Per_Hertz_Overfluxing_Trip := FALSE;
    Generator_Loss_of_Field_Trip := FALSE;
    Field_Overcurrent_Trip_Latched := FALSE;
END_IF;

(* 1. Volts-per-Hertz (Overfluxing) Protection: V / Hz ratio check *)
(* Ratio = (V / 138) / (Hz / 6000) * 100 *)
IF (Generator_Frequency_Hz > 1000) THEN
    IF ((Generator_Terminal_Voltage_kV * 6000) / (Generator_Frequency_Hz * 138) * 100) >= V_Per_Hz_Limit_Ratio THEN
        Volts_Per_Hertz_Overfluxing_Trip := TRUE;
    END_IF;
END_IF;

(* 2. Loss of Field (40 Relay) Protection *)
IF Generator_Breaker_Closed AND (Generator_Reactive_Power_MVAR <= Loss_of_Field_Threshold_MVAR) AND (Excitation_Field_Current_Amps < 50) THEN
    Generator_Loss_of_Field_Trip := TRUE;
END_IF;

(* 3. Field Overcurrent Protection *)
IF Excitation_Field_Current_Amps >= 850 THEN
    Field_Overcurrent_Trip_Latched := TRUE;
END_IF;

(* 4. Active Trip Enforcement *)
IF Volts_Per_Hertz_Overfluxing_Trip OR Generator_Loss_of_Field_Trip OR Field_Overcurrent_Trip_Latched THEN
    Field_Breaker_Close_Command := FALSE;
    AVR_Automatic_Mode_Active := FALSE;
    Under_Excitation_Limiter_Active := FALSE;
    Over_Excitation_Limiter_Active := FALSE;
    Excitation_Field_Voltage_Volts := 0;
ELSE
    Field_Breaker_Close_Command := TRUE;
    IF AVR_Auto_Select THEN
        AVR_Automatic_Mode_Active := TRUE;

        (* 5. Over-Excitation Limiter (OEL) *)
        IF Excitation_Field_Current_Amps >= OEL_Threshold_Amps THEN
            Over_Excitation_Limiter_Active := TRUE;
            Excitation_Field_Voltage_Volts := 140;
        ELSE
            Over_Excitation_Limiter_Active := FALSE;
        END_IF;

        (* 6. Under-Excitation Limiter (UEL) *)
        IF Generator_Reactive_Power_MVAR <= UEL_Threshold_MVAR THEN
            Under_Excitation_Limiter_Active := TRUE;
            Excitation_Field_Voltage_Volts := 110;
        ELSE
            Under_Excitation_Limiter_Active := FALSE;
        END_IF;

        (* Normal AVR closed-loop voltage regulation *)
        IF NOT Over_Excitation_Limiter_Active AND NOT Under_Excitation_Limiter_Active THEN
            Excitation_Field_Voltage_Volts := 125;
        END_IF;
    ELSE
        AVR_Automatic_Mode_Active := FALSE;
    END_IF;
END_IF;

END_FUNCTION_BLOCK

(* ---- lead_lag_pump_controller.st ---- *)
(* ============================================================================
 * Title:       FB_LeadLagPumpControl
 * Description: Industrial Duplex Lead-Lag Alternating Pump Controller.
 * Features:
 *   - Automatic wear-leveling duty/standby rotation based on run hours
 *   - Auto-switchover on pump trip, overload, or dry-run fault
 *   - Lag pump staging when process demand exceeds single pump capacity
 *   - Anti-short-cycling minimum run and minimum rest timers
 *   - Independent Hand/Off/Auto operation with maintenance warning thresholds
 * Language:    IEC 61131-3 Structured Text (Pure ST)
 * ============================================================================ *)

FUNCTION_BLOCK FB_LeadLagPumpControl
VAR_INPUT
    AutoEnable : BOOL := TRUE;            (* Master automatic control permissive *)
    DemandLevel : REAL := 0.0;            (* Current wet-well level or process demand (0.0 to 100.0 %) *)
    LeadStartSP : REAL := 60.0;           (* Level threshold to start lead pump (%) *)
    LagStartSP : REAL := 85.0;            (* Level threshold to stage in lag pump (%) *)
    StopSP : REAL := 20.0;                (* Level threshold to stop all pumps (%) *)
    Pump1_Tripped : BOOL := FALSE;        (* Pump 1 thermal overload / drive fault *)
    Pump2_Tripped : BOOL := FALSE;        (* Pump 2 thermal overload / drive fault *)
    Pump1_DryRun : BOOL := FALSE;         (* Pump 1 low suction / dry run sensor *)
    Pump2_DryRun : BOOL := FALSE;         (* Pump 2 low suction / dry run sensor *)
    ManualMode : BOOL := FALSE;           (* Manual override select: TRUE = Manual, FALSE = Auto *)
    Pump1_Manual : BOOL := FALSE;         (* Manual start command for Pump 1 *)
    Pump2_Manual : BOOL := FALSE;         (* Manual start command for Pump 2 *)
    ResetFaults : BOOL := FALSE;          (* Latch clear / fault reset push button *)
    MaxRuntimeHours : REAL := 5000.0;     (* Preventive maintenance hour threshold *)
    MinRunTimeSec : REAL := 15.0;         (* Minimum run duration to prevent short cycling *)
    MinRestTimeSec : REAL := 20.0;        (* Minimum rest delay before motor re-start *)
    CycleTimeSec : REAL := 0.1;           (* PLC cyclic task scan period (seconds) *)
END_VAR

VAR_OUTPUT
    Pump1_RunCmd : BOOL := FALSE;         (* Digital output: Pump 1 contactor / VFD run *)
    Pump2_RunCmd : BOOL := FALSE;         (* Digital output: Pump 2 contactor / VFD run *)
    LeadPumpId : INT := 1;                (* Currently designated lead pump (1 or 2) *)
    LagActive : BOOL := FALSE;            (* TRUE when secondary lag pump is commanded *)
    Pump1_Hours : REAL := 0.0;            (* Accumulated running hours on Pump 1 *)
    Pump2_Hours : REAL := 0.0;            (* Accumulated running hours on Pump 2 *)
    Pump1_Starts : DINT := 0;             (* Total start cycles on Pump 1 *)
    Pump2_Starts : DINT := 0;             (* Total start cycles on Pump 2 *)
    Pump1_Fault : BOOL := FALSE;          (* Latched fault status for Pump 1 *)
    Pump2_Fault : BOOL := FALSE;          (* Latched fault status for Pump 2 *)
    AllPumpsFaulted : BOOL := FALSE;      (* Alarm: No pumps available to service demand *)
    ServiceReqPump1 : BOOL := FALSE;      (* Maintenance warning: Pump 1 runtime exceeded *)
    ServiceReqPump2 : BOOL := FALSE;      (* Maintenance warning: Pump 2 runtime exceeded *)
END_VAR

VAR
    P1_RunTimer : REAL := 0.0;            (* Seconds Pump 1 has run in current cycle *)
    P2_RunTimer : REAL := 0.0;            (* Seconds Pump 2 has run in current cycle *)
    P1_RestTimer : REAL := 30.0;          (* Seconds Pump 1 has rested since last stop *)
    P2_RestTimer : REAL := 30.0;          (* Seconds Pump 2 has rested since last stop *)
    P1_PrevRun : BOOL := FALSE;           (* Rising edge detection for starts counter *)
    P2_PrevRun : BOOL := FALSE;           (* Rising edge detection for starts counter *)
    P1_Available : BOOL := TRUE;          (* Pump 1 ready for service *)
    P2_Available : BOOL := TRUE;          (* Pump 2 ready for service *)
    DemandActive : BOOL := FALSE;         (* Process level demand state *)
    LagDemandActive : BOOL := FALSE;      (* High demand requiring both pumps *)
END_VAR

(* 1. Fault Evaluation and Latching *)
IF ResetFaults THEN
    Pump1_Fault := FALSE;
    Pump2_Fault := FALSE;
END_IF;

IF Pump1_Tripped OR Pump1_DryRun THEN
    Pump1_Fault := TRUE;
END_IF;

IF Pump2_Tripped OR Pump2_DryRun THEN
    Pump2_Fault := TRUE;
END_IF;

P1_Available := NOT Pump1_Fault;
P2_Available := NOT Pump2_Fault;
AllPumpsFaulted := (NOT P1_Available) AND (NOT P2_Available);

(* 2. Process Demand Hysteresis Evaluation *)
IF DemandLevel >= LeadStartSP THEN
    DemandActive := TRUE;
ELSIF DemandLevel <= StopSP THEN
    DemandActive := FALSE;
END_IF;

IF DemandLevel >= LagStartSP THEN
    LagDemandActive := TRUE;
ELSIF DemandLevel < LeadStartSP THEN
    LagDemandActive := FALSE;
END_IF;

(* 3. Lead Selection & Wear Leveling *)
(* Rotate lead assignment when both pumps are off or if lead pump faults *)
IF (NOT Pump1_RunCmd) AND (NOT Pump2_RunCmd) THEN
    IF P1_Available AND P2_Available THEN
        IF Pump1_Hours <= Pump2_Hours THEN
            LeadPumpId := 1;
        ELSE
            LeadPumpId := 2;
        END_IF;
    ELSIF P1_Available THEN
        LeadPumpId := 1;
    ELSIF P2_Available THEN
        LeadPumpId := 2;
    END_IF;
ELSIF LeadPumpId = 1 AND (NOT P1_Available) AND P2_Available THEN
    (* Immediate auto-switchover upon lead pump failure *)
    LeadPumpId := 2;
ELSIF LeadPumpId = 2 AND (NOT P2_Available) AND P1_Available THEN
    (* Immediate auto-switchover upon lead pump failure *)
    LeadPumpId := 1;
END_IF;

(* 4. Automatic / Manual Control Execution *)
IF ManualMode THEN
    (* Manual Hand Mode *)
    Pump1_RunCmd := Pump1_Manual AND P1_Available;
    Pump2_RunCmd := Pump2_Manual AND P2_Available;
    LagActive := Pump1_RunCmd AND Pump2_RunCmd;
ELSIF AutoEnable AND (NOT AllPumpsFaulted) THEN
    (* Automatic Duplex Control *)
    IF DemandActive THEN
        IF LeadPumpId = 1 THEN
            (* Pump 1 is Lead *)
            IF P1_Available AND (P1_RestTimer >= MinRestTimeSec OR Pump1_RunCmd) THEN
                Pump1_RunCmd := TRUE;
            ELSE
                Pump1_RunCmd := FALSE;
            END_IF;

            (* Pump 2 is Lag *)
            IF LagDemandActive OR (NOT P1_Available) THEN
                IF P2_Available AND (P2_RestTimer >= MinRestTimeSec OR Pump2_RunCmd) THEN
                    Pump2_RunCmd := TRUE;
                ELSE
                    Pump2_RunCmd := FALSE;
                END_IF;
            ELSE
                IF P2_RunTimer >= MinRunTimeSec THEN
                    Pump2_RunCmd := FALSE;
                END_IF;
            END_IF;
        ELSE
            (* Pump 2 is Lead *)
            IF P2_Available AND (P2_RestTimer >= MinRestTimeSec OR Pump2_RunCmd) THEN
                Pump2_RunCmd := TRUE;
            ELSE
                Pump2_RunCmd := FALSE;
            END_IF;

            (* Pump 1 is Lag *)
            IF LagDemandActive OR (NOT P2_Available) THEN
                IF P1_Available AND (P1_RestTimer >= MinRestTimeSec OR Pump1_RunCmd) THEN
                    Pump1_RunCmd := TRUE;
                ELSE
                    Pump1_RunCmd := FALSE;
                END_IF;
            ELSE
                IF P1_RunTimer >= MinRunTimeSec THEN
                    Pump1_RunCmd := FALSE;
                END_IF;
            END_IF;
        END_IF;
    ELSE
        (* Below stop setpoint: respect minimum run time before stopping *)
        IF P1_RunTimer >= MinRunTimeSec THEN
            Pump1_RunCmd := FALSE;
        END_IF;
        IF P2_RunTimer >= MinRunTimeSec THEN
            Pump2_RunCmd := FALSE;
        END_IF;
    END_IF;

    LagActive := Pump1_RunCmd AND Pump2_RunCmd;
ELSE
    (* System disabled or critical lockout *)
    Pump1_RunCmd := FALSE;
    Pump2_RunCmd := FALSE;
    LagActive := FALSE;
END_IF;

(* Safety interlock override: faulted pumps are unconditionally prohibited from running *)
IF NOT P1_Available THEN
    Pump1_RunCmd := FALSE;
END_IF;
IF NOT P2_Available THEN
    Pump2_RunCmd := FALSE;
END_IF;
LagActive := Pump1_RunCmd AND Pump2_RunCmd;

(* 5. Runtime, Rest-Time, and Cycle Accumulation *)
IF Pump1_RunCmd THEN
    P1_RunTimer := P1_RunTimer + CycleTimeSec;
    P1_RestTimer := 0.0;
    Pump1_Hours := Pump1_Hours + (CycleTimeSec / 3600.0);
    IF NOT P1_PrevRun THEN
        Pump1_Starts := Pump1_Starts + 1;
    END_IF;
ELSE
    P1_RunTimer := 0.0;
    P1_RestTimer := P1_RestTimer + CycleTimeSec;
END_IF;
P1_PrevRun := Pump1_RunCmd;

IF Pump2_RunCmd THEN
    P2_RunTimer := P2_RunTimer + CycleTimeSec;
    P2_RestTimer := 0.0;
    Pump2_Hours := Pump2_Hours + (CycleTimeSec / 3600.0);
    IF NOT P2_PrevRun THEN
        Pump2_Starts := Pump2_Starts + 1;
    END_IF;
ELSE
    P2_RunTimer := 0.0;
    P2_RestTimer := P2_RestTimer + CycleTimeSec;
END_IF;
P2_PrevRun := Pump2_RunCmd;

(* 6. Preventive Maintenance Hour Warnings *)
ServiceReqPump1 := Pump1_Hours >= MaxRuntimeHours;
ServiceReqPump2 := Pump2_Hours >= MaxRuntimeHours;

END_FUNCTION_BLOCK

(* ---- pid_temperature_controller.st ---- *)
(* ============================================================================
 * Title:       FB_PIDTemperatureControl
 * Description: Industrial Closed-Loop Precision Temperature PID Controller.
 * Features:
 *   - First-order low-pass noise filter on raw process variable (PV)
 *   - Proportional-Integral-Derivative algorithm with Anti-Reset Windup
 *   - Derivative on PV action to eliminate setpoint change kicks
 *   - Bumpless transfer between Manual and Automatic modes
 *   - Deadband gap to eliminate unnecessary actuator hunting
 *   - Time-proportional PWM output for solid-state relay (SSR) heating
 *   - Analog modulating cooling output (split-range heat/cool control)
 *   - Multi-tier process safety alarms: High-High, High, Low, Low-Low
 * Language:    IEC 61131-3 Structured Text (Pure ST)
 * ============================================================================ *)

FUNCTION_BLOCK FB_PIDTemperatureControl
VAR_INPUT
    Enable : BOOL := TRUE;                (* Master loop enable permissive *)
    Setpoint : REAL := 150.0;             (* Desired temperature setpoint in Deg C *)
    RawPV : REAL := 25.0;                 (* Unfiltered process variable from analog input *)
    ManualMode : BOOL := FALSE;           (* Mode select: TRUE = Manual, FALSE = Auto PID *)
    ManualOutput : REAL := 0.0;           (* Manual output target (0.0 to 100.0 %) *)
    Kp : REAL := 4.5;                     (* Proportional gain *)
    Ki : REAL := 0.05;                    (* Integral gain (1 / second) *)
    Kd : REAL := 1.20;                    (* Derivative gain (seconds) *)
    Deadband : REAL := 0.5;               (* Error deadband zone (+/- Deg C) *)
    FilterAlpha : REAL := 0.25;           (* PV 1st-order filter coefficient (0.01 to 1.0) *)
    CycleTimeSec : REAL := 0.1;           (* Scan period of the calling task (seconds) *)
    PwmPeriodSec : REAL := 5.0;           (* Time-proportional SSR heating cycle base (seconds) *)
    SplitRangeMid : REAL := 50.0;         (* Split-range boundary between cool and heat (%) *)
    HighHighSP : REAL := 220.0;           (* Emergency High-High temperature trip point *)
    HighSP : REAL := 180.0;               (* High temperature warning setpoint *)
    LowSP : REAL := 80.0;                 (* Low temperature warning setpoint *)
    LowLowSP : REAL := 50.0;              (* Critical Low-Low temperature trip point *)
    SensorFault : BOOL := FALSE;          (* Open thermocouple / RTD wire-break signal *)
    ResetAlarm : BOOL := FALSE;           (* Alarm acknowledgment / reset input *)
END_VAR

VAR_OUTPUT
    HeatOutput : REAL := 0.0;             (* Modulating heating demand (0.0 to 100.0 %) *)
    CoolOutput : REAL := 0.0;             (* Modulating cooling demand (0.0 to 100.0 %) *)
    PWM_Heater : BOOL := FALSE;           (* Digital pulse to SSR / contactor *)
    FilteredPV : REAL := 25.0;            (* Noise-filtered process temperature *)
    Error : REAL := 0.0;                  (* Regulation error (Setpoint - FilteredPV) *)
    AlarmHH : BOOL := FALSE;              (* Latched High-High critical trip alarm *)
    AlarmH : BOOL := FALSE;               (* High temperature warning alarm *)
    AlarmL : BOOL := FALSE;               (* Low temperature warning alarm *)
    AlarmLL : BOOL := FALSE;              (* Latched Low-Low critical trip alarm *)
    LoopHealthy : BOOL := TRUE;           (* Operational health status of loop *)
END_VAR

VAR
    LastPV : REAL := 25.0;                (* Previous PV for derivative computation *)
    IntegralSum : REAL := 0.0;            (* Accumulated integral sum *)
    PropTerm : REAL := 0.0;               (* Calculated proportional contribution *)
    DerivTerm : REAL := 0.0;              (* Calculated derivative contribution *)
    TotalEffort : REAL := 0.0;            (* Net unclamped control output (0.0 to 100.0 %) *)
    EffectiveError : REAL := 0.0;         (* Error after deadband filtering *)
    PwmAccumulator : REAL := 0.0;         (* Accumulator for PWM period generator *)
END_VAR

(* 1. Alarm Reset and Sensor Fault Evaluation *)
IF ResetAlarm THEN
    AlarmHH := FALSE;
    AlarmLL := FALSE;
END_IF;

IF SensorFault THEN
    LoopHealthy := FALSE;
    HeatOutput := 0.0;
    CoolOutput := 0.0;
    PWM_Heater := FALSE;
    RETURN;
END_IF;

(* 2. First-Order Digital Low-Pass Noise Filter on PV *)
FilteredPV := (FilterAlpha * RawPV) + ((1.0 - FilterAlpha) * FilteredPV);

(* 3. Process Safety Alarms *)
IF FilteredPV >= HighHighSP THEN
    AlarmHH := TRUE;
END_IF;

IF FilteredPV <= LowLowSP THEN
    AlarmLL := TRUE;
END_IF;

AlarmH := FilteredPV >= HighSP;
AlarmL := FilteredPV <= LowSP;
LoopHealthy := (NOT AlarmHH) AND (NOT SensorFault);

(* 4. Error Calculation with Deadband *)
Error := Setpoint - FilteredPV;

IF ABS(Error) <= Deadband THEN
    EffectiveError := 0.0;
ELSE
    EffectiveError := Error;
END_IF;

(* 5. Auto / Manual PID Algorithm *)
IF (NOT Enable) OR AlarmHH THEN
    (* Safety shutdown state *)
    HeatOutput := 0.0;
    CoolOutput := 0.0;
    IntegralSum := 0.0;
    TotalEffort := 0.0;
    LastPV := FilteredPV;
ELSIF ManualMode THEN
    (* Manual Override Mode with Bumpless Tracking *)
    TotalEffort := LIMIT(0.0, ManualOutput, 100.0);
    IntegralSum := TotalEffort;
    LastPV := FilteredPV;

    IF TotalEffort >= SplitRangeMid THEN
        HeatOutput := (TotalEffort - SplitRangeMid) * (100.0 / (100.0 - SplitRangeMid));
        CoolOutput := 0.0;
    ELSE
        HeatOutput := 0.0;
        CoolOutput := (SplitRangeMid - TotalEffort) * (100.0 / SplitRangeMid);
    END_IF;
ELSE
    (* Automatic PID Regulation *)
    (* Proportional Term *)
    PropTerm := Kp * EffectiveError;

    (* Integral Term with Anti-Reset Windup *)
    IntegralSum := IntegralSum + (Ki * EffectiveError * CycleTimeSec);
    IntegralSum := LIMIT(0.0, IntegralSum, 100.0);

    (* Derivative on Measurement: -Kd * d(PV)/dt eliminates setpoint kick *)
    DerivTerm := -1.0 * Kd * (FilteredPV - LastPV) / CycleTimeSec;
    LastPV := FilteredPV;

    (* Total Control Output [0.0 to 100.0 %] *)
    TotalEffort := LIMIT(0.0, PropTerm + IntegralSum + DerivTerm, 100.0);

    (* Split-Range Actuation (Heat / Cool) *)
    IF TotalEffort >= SplitRangeMid THEN
        HeatOutput := (TotalEffort - SplitRangeMid) * (100.0 / (100.0 - SplitRangeMid));
        CoolOutput := 0.0;
    ELSE
        HeatOutput := 0.0;
        CoolOutput := (SplitRangeMid - TotalEffort) * (100.0 / SplitRangeMid);
    END_IF;
END_IF;

(* 6. Time-Proportional PWM Solid-State Relay Generation *)
IF Enable AND (NOT AlarmHH) AND (HeatOutput > 0.0) THEN
    PwmAccumulator := PwmAccumulator + (CycleTimeSec / PwmPeriodSec * 100.0);
    IF PwmAccumulator >= 100.0 THEN
        PwmAccumulator := 0.0;
    END_IF;
    PWM_Heater := PwmAccumulator < HeatOutput;
ELSE
    PwmAccumulator := 0.0;
    PWM_Heater := FALSE;
END_IF;

END_FUNCTION_BLOCK

(* ---- pump_lead_lag_alternator.st ---- *)
(* ============================================================================
 * Title:       FB_PumpLeadLagAlternator
 * Description: Industrial Duplex Lead-Lag Alternating Pump Controller with
 *              Wear-Leveling, Sub-Second Failover, Dual-Pump Boost, and
 *              Anti-Hunting Debounce Timers.
 * Features:
 *   - Lead/Lag pump duty alternation based on accumulated runtime hours (%R151, %R152)
 *   - Automatic sub-second failover to standby pump if lead pump trips or faults (%M83, %M84)
 *   - High-demand dual-pump boost mode when system pressure falls below low setpoint
 *   - Manual pump force/override switches for maintenance
 *   - Pump start/stop anti-hunting debouncing and minimum run/rest timers
 * Language:    IEC 61131-3 Structured Text (Pure ST Only)
 * OCS Mapping:
 *   %R151: Pump1_Runtime_Hours (REAL: Accumulated runtime hours for Pump 1)
 *   %R152: Pump2_Runtime_Hours (REAL: Accumulated runtime hours for Pump 2)
 *   %R153: System_Pressure_PSI (REAL: Current system discharge header pressure)
 *   %R154: Lead_Start_SP (REAL: Pressure threshold to start lead pump)
 *   %R155: Boost_Start_SP (REAL: Pressure threshold for dual-pump boost mode)
 *   %R156: Stop_SP (REAL: Pressure threshold to stop pumps)
 *   %M81:  Manual_Mode_Select (BOOL: TRUE = Manual, FALSE = Auto)
 *   %M82:  Auto_Enable (BOOL: Master automatic staging permissive)
 *   %M83:  Pump1_Trip_Fault (BOOL: Pump 1 thermal overload / drive trip)
 *   %M84:  Pump2_Trip_Fault (BOOL: Pump 2 thermal overload / drive trip)
 *   %M85:  Pump1_Manual_Override (BOOL: Manual force run command for Pump 1)
 *   %M86:  Pump2_Manual_Override (BOOL: Manual force run command for Pump 2)
 *   %M87:  Pump1_Lockout (BOOL: Maintenance lockout switch for Pump 1)
 *   %M88:  Pump2_Lockout (BOOL: Maintenance lockout switch for Pump 2)
 *   %M89:  Fault_Reset (BOOL: Latch clear / fault reset push button)
 *   %Q51:  Pump1_Run_Cmd (BOOL: Digital output contactor / VFD run for Pump 1)
 *   %Q52:  Pump2_Run_Cmd (BOOL: Digital output contactor / VFD run for Pump 2)
 *   %M91:  Boost_Mode_Active (BOOL: Dual-pump boost mode active)
 *   %M92:  Failover_Active (BOOL: Sub-second failover active)
 * ============================================================================ *)

FUNCTION_BLOCK FB_PumpLeadLagAlternator
VAR_INPUT
    Auto_Enable : BOOL := TRUE;                    (* Master automatic staging permissive (%M82) *)
    System_Pressure_PSI : REAL := 55.0;            (* System header pressure measurement (%R153) *)
    Lead_Start_SP : REAL := 45.0;                  (* Header pressure threshold to start lead pump (%R154) *)
    Boost_Start_SP : REAL := 35.0;                 (* Low pressure threshold for dual-pump boost mode (%R155) *)
    Stop_SP : REAL := 60.0;                        (* High pressure threshold to stop running pumps (%R156) *)
    Pump1_Trip_Fault : BOOL := FALSE;              (* Pump 1 thermal overload / drive trip (%M83) *)
    Pump2_Trip_Fault : BOOL := FALSE;              (* Pump 2 thermal overload / drive trip (%M84) *)
    Manual_Mode_Select : BOOL := FALSE;            (* Mode selector: TRUE = Manual Hand, FALSE = Auto (%M81) *)
    Pump1_Manual_Override : BOOL := FALSE;         (* Manual force run switch for Pump 1 (%M85) *)
    Pump2_Manual_Override : BOOL := FALSE;         (* Manual force run switch for Pump 2 (%M86) *)
    Pump1_Lockout : BOOL := FALSE;                 (* Maintenance lockout switch for Pump 1 (%M87) *)
    Pump2_Lockout : BOOL := FALSE;                 (* Maintenance lockout switch for Pump 2 (%M88) *)
    Fault_Reset : BOOL := FALSE;                   (* Latch clear / fault reset push button (%M89) *)
    Debounce_Time_Sec : REAL := 2.0;               (* Anti-hunting pressure qualification debounce delay *)
    Min_Run_Time_Sec : REAL := 15.0;               (* Minimum run time to prevent short cycling *)
    Min_Rest_Time_Sec : REAL := 20.0;              (* Minimum resting delay before motor restart *)
    Cycle_Time_Sec : REAL := 0.1;                  (* Scan execution period in seconds *)
END_VAR

VAR_OUTPUT
    Pump1_Run_Cmd : BOOL := FALSE;                 (* Command contactor / VFD run for Pump 1 (%Q51) *)
    Pump2_Run_Cmd : BOOL := FALSE;                 (* Command contactor / VFD run for Pump 2 (%Q52) *)
    Lead_Pump_Id : INT := 1;                       (* Current lead pump assignment (1 or 2) *)
    Lag_Pump_Id : INT := 2;                        (* Current lag / standby pump assignment (1 or 2) *)
    Boost_Mode_Active : BOOL := FALSE;             (* Dual-pump boost mode active due to high demand (%M91) *)
    Failover_Active : BOOL := FALSE;               (* Sub-second failover active due to lead pump trip (%M92) *)
    Pump1_Runtime_Hours : REAL := 0.0;             (* Accumulated running hours for Pump 1 (%R151) *)
    Pump2_Runtime_Hours : REAL := 0.0;             (* Accumulated running hours for Pump 2 (%R152) *)
    Pump1_Starts_Count : DINT := 0;                (* Total start cycles on Pump 1 *)
    Pump2_Starts_Count : DINT := 0;                (* Total start cycles on Pump 2 *)
    Pump1_Fault_Latched : BOOL := FALSE;           (* Latched trip status for Pump 1 *)
    Pump2_Fault_Latched : BOOL := FALSE;           (* Latched trip status for Pump 2 *)
    System_Fault_Alarm : BOOL := FALSE;            (* Alarm: No healthy pumps available to service demand *)
END_VAR

VAR
    P1_Run_Timer : REAL := 0.0;                    (* Current cycle run timer for Pump 1 *)
    P2_Run_Timer : REAL := 0.0;                    (* Current cycle run timer for Pump 2 *)
    P1_Rest_Timer : REAL := 30.0;                  (* Time elapsed since Pump 1 stopped *)
    P2_Rest_Timer : REAL := 30.0;                  (* Time elapsed since Pump 2 stopped *)
    Lead_Debounce_Timer : REAL := 0.0;             (* Accumulator for lead start debounce *)
    Boost_Debounce_Timer : REAL := 0.0;            (* Accumulator for boost start debounce *)
    Stop_Debounce_Timer : REAL := 0.0;             (* Accumulator for stop debounce *)
    P1_Prev_Run : BOOL := FALSE;                   (* Previous scan run state for edge detection *)
    P2_Prev_Run : BOOL := FALSE;                   (* Previous scan run state for edge detection *)
    Lead_Req_Debounced : BOOL := FALSE;            (* Anti-hunting debounced lead start demand *)
    Boost_Req_Debounced : BOOL := FALSE;           (* Anti-hunting debounced boost start demand *)
    Stop_Req_Debounced : BOOL := FALSE;            (* Anti-hunting debounced stop demand *)
    P1_Available : BOOL := TRUE;                   (* Pump 1 ready and healthy *)
    P2_Available : BOOL := TRUE;                   (* Pump 2 ready and healthy *)
END_VAR

(* 1. Fault Handling and Maintenance Lockout *)
IF Fault_Reset THEN
    Pump1_Fault_Latched := FALSE;
    Pump2_Fault_Latched := FALSE;
    Failover_Active := FALSE;
END_IF;

IF Pump1_Trip_Fault THEN
    Pump1_Fault_Latched := TRUE;
END_IF;

IF Pump2_Trip_Fault THEN
    Pump2_Fault_Latched := TRUE;
END_IF;

P1_Available := (NOT Pump1_Fault_Latched) AND (NOT Pump1_Lockout);
P2_Available := (NOT Pump2_Fault_Latched) AND (NOT Pump2_Lockout);
System_Fault_Alarm := (NOT P1_Available) AND (NOT P2_Available);

(* 2. Anti-Hunting Pressure Signal Debouncing *)
IF System_Pressure_PSI <= Lead_Start_SP THEN
    Lead_Debounce_Timer := Lead_Debounce_Timer + Cycle_Time_Sec;
    IF Lead_Debounce_Timer >= Debounce_Time_Sec THEN
        Lead_Req_Debounced := TRUE;
    END_IF;
ELSE
    Lead_Debounce_Timer := 0.0;
END_IF;

IF System_Pressure_PSI <= Boost_Start_SP THEN
    Boost_Debounce_Timer := Boost_Debounce_Timer + Cycle_Time_Sec;
    IF Boost_Debounce_Timer >= Debounce_Time_Sec THEN
        Boost_Req_Debounced := TRUE;
    END_IF;
ELSE
    Boost_Debounce_Timer := 0.0;
    Boost_Req_Debounced := FALSE;
END_IF;

IF System_Pressure_PSI >= Stop_SP THEN
    Stop_Debounce_Timer := Stop_Debounce_Timer + Cycle_Time_Sec;
    IF Stop_Debounce_Timer >= Debounce_Time_Sec THEN
        Stop_Req_Debounced := TRUE;
        Lead_Req_Debounced := FALSE;
        Boost_Req_Debounced := FALSE;
    END_IF;
ELSE
    Stop_Debounce_Timer := 0.0;
    Stop_Req_Debounced := FALSE;
END_IF;

(* 3. Lead/Lag Alternation and Sub-Second Failover *)
IF (NOT Pump1_Run_Cmd) AND (NOT Pump2_Run_Cmd) THEN
    IF P1_Available AND P2_Available THEN
        IF Pump1_Runtime_Hours <= Pump2_Runtime_Hours THEN
            Lead_Pump_Id := 1;
            Lag_Pump_Id := 2;
        ELSE
            Lead_Pump_Id := 2;
            Lag_Pump_Id := 1;
        END_IF;
    ELSIF P1_Available THEN
        Lead_Pump_Id := 1;
        Lag_Pump_Id := 2;
    ELSIF P2_Available THEN
        Lead_Pump_Id := 2;
        Lag_Pump_Id := 1;
    END_IF;
ELSIF Lead_Pump_Id = 1 AND (NOT P1_Available) AND P2_Available THEN
    Lead_Pump_Id := 2;
    Lag_Pump_Id := 1;
    Failover_Active := TRUE;
ELSIF Lead_Pump_Id = 2 AND (NOT P2_Available) AND P1_Available THEN
    Lead_Pump_Id := 1;
    Lag_Pump_Id := 2;
    Failover_Active := TRUE;
END_IF;

(* 4. Automatic / Manual Control Execution with Minimum Run/Rest Timers *)
IF Manual_Mode_Select THEN
    Pump1_Run_Cmd := Pump1_Manual_Override AND P1_Available;
    Pump2_Run_Cmd := Pump2_Manual_Override AND P2_Available;
    Boost_Mode_Active := Pump1_Run_Cmd AND Pump2_Run_Cmd;
ELSIF Auto_Enable AND (NOT System_Fault_Alarm) THEN
    IF Lead_Req_Debounced THEN
        IF Lead_Pump_Id = 1 THEN
            IF P1_Available AND (P1_Rest_Timer >= Min_Rest_Time_Sec OR Pump1_Run_Cmd) THEN
                Pump1_Run_Cmd := TRUE;
            ELSE
                Pump1_Run_Cmd := FALSE;
            END_IF;

            IF Boost_Req_Debounced OR Failover_Active OR (NOT P1_Available) THEN
                IF P2_Available AND (P2_Rest_Timer >= Min_Rest_Time_Sec OR Pump2_Run_Cmd) THEN
                    Pump2_Run_Cmd := TRUE;
                ELSE
                    Pump2_Run_Cmd := FALSE;
                END_IF;
            ELSE
                IF P2_Run_Timer >= Min_Run_Time_Sec THEN
                    Pump2_Run_Cmd := FALSE;
                END_IF;
            END_IF;
        ELSE
            IF P2_Available AND (P2_Rest_Timer >= Min_Rest_Time_Sec OR Pump2_Run_Cmd) THEN
                Pump2_Run_Cmd := TRUE;
            ELSE
                Pump2_Run_Cmd := FALSE;
            END_IF;

            IF Boost_Req_Debounced OR Failover_Active OR (NOT P2_Available) THEN
                IF P1_Available AND (P1_Rest_Timer >= Min_Rest_Time_Sec OR Pump1_Run_Cmd) THEN
                    Pump1_Run_Cmd := TRUE;
                ELSE
                    Pump1_Run_Cmd := FALSE;
                END_IF;
            ELSE
                IF P1_Run_Timer >= Min_Run_Time_Sec THEN
                    Pump1_Run_Cmd := FALSE;
                END_IF;
            END_IF;
        END_IF;
    ELSIF Stop_Req_Debounced THEN
        IF P1_Run_Timer >= Min_Run_Time_Sec THEN
            Pump1_Run_Cmd := FALSE;
        END_IF;
        IF P2_Run_Timer >= Min_Run_Time_Sec THEN
            Pump2_Run_Cmd := FALSE;
        END_IF;
    END_IF;

    Boost_Mode_Active := Pump1_Run_Cmd AND Pump2_Run_Cmd;
ELSE
    Pump1_Run_Cmd := FALSE;
    Pump2_Run_Cmd := FALSE;
    Boost_Mode_Active := FALSE;
END_IF;

(* Safety interlock override: unavailable pumps cannot run *)
IF NOT P1_Available THEN
    Pump1_Run_Cmd := FALSE;
END_IF;
IF NOT P2_Available THEN
    Pump2_Run_Cmd := FALSE;
END_IF;
Boost_Mode_Active := Pump1_Run_Cmd AND Pump2_Run_Cmd;

(* 5. Runtime, Rest-Time, and Cycle Accumulation *)
IF Pump1_Run_Cmd THEN
    P1_Run_Timer := P1_Run_Timer + Cycle_Time_Sec;
    P1_Rest_Timer := 0.0;
    Pump1_Runtime_Hours := Pump1_Runtime_Hours + (Cycle_Time_Sec / 3600.0);
    IF NOT P1_Prev_Run THEN
        Pump1_Starts_Count := Pump1_Starts_Count + 1;
    END_IF;
ELSE
    P1_Run_Timer := 0.0;
    P1_Rest_Timer := P1_Rest_Timer + Cycle_Time_Sec;
END_IF;
P1_Prev_Run := Pump1_Run_Cmd;

IF Pump2_Run_Cmd THEN
    P2_Run_Timer := P2_Run_Timer + Cycle_Time_Sec;
    P2_Rest_Timer := 0.0;
    Pump2_Runtime_Hours := Pump2_Runtime_Hours + (Cycle_Time_Sec / 3600.0);
    IF NOT P2_Prev_Run THEN
        Pump2_Starts_Count := Pump2_Starts_Count + 1;
    END_IF;
ELSE
    P2_Run_Timer := 0.0;
    P2_Rest_Timer := P2_Rest_Timer + Cycle_Time_Sec;
END_IF;
P2_Prev_Run := Pump2_Run_Cmd;

END_FUNCTION_BLOCK

(* ---- ramp_rate_limiter.st ---- *)
(* ============================================================================
 * Title:       FB_RampRateLimiter
 * Description: Industrial Setpoint Slew-Rate Limiter & Motion Profiler.
 * Features:
 *   - Independent acceleration (Ramp Up) and deceleration (Ramp Down) rate limits
 *   - Smooth, linear setpoint profiling to prevent mechanical or thermal stress
 *   - Anti-overshoot clamping directly to target value
 *   - Instantaneous bypass mode for emergency positioning or step jumps
 *   - Target reached status and active direction indicators
 * Language:    IEC 61131-3 Structured Text (Pure ST)
 * ============================================================================ *)

FUNCTION_BLOCK FB_RampRateLimiter
VAR_INPUT
    TargetValue : REAL := 0.0;            (* Desired target setpoint in Engineering Units *)
    RampUpRate : REAL := 10.0;            (* Maximum allowable rate of increase (EU / second) *)
    RampDownRate : REAL := 10.0;          (* Maximum allowable rate of decrease (EU / second) *)
    BypassRamp : BOOL := FALSE;           (* TRUE = immediate step jump to TargetValue *)
    InitCmd : BOOL := FALSE;              (* Force output to InitValue *)
    InitValue : REAL := 0.0;              (* Preload value when InitCmd is active *)
    Deadband : REAL := 0.01;              (* Threshold band for declaring target reached *)
    CycleTimeSec : REAL := 0.1;           (* Execution scan period (seconds) *)
END_VAR

VAR_OUTPUT
    CurrentValue : REAL := 0.0;           (* Output following rate-limited profile *)
    RampingUp : BOOL := FALSE;            (* TRUE while output is ascending toward target *)
    RampingDown : BOOL := FALSE;          (* TRUE while output is descending toward target *)
    TargetReached : BOOL := TRUE;         (* TRUE when output is within Deadband of target *)
    DeltaRate : REAL := 0.0;              (* Actual rate of change applied (EU / second) *)
END_VAR

VAR
    MaxUpStep : REAL := 0.0;              (* Maximum positive change per cycle *)
    MaxDownStep : REAL := 0.0;            (* Maximum negative change per cycle *)
    Difference : REAL := 0.0;             (* Distance from target (TargetValue - CurrentValue) *)
    PrevValue : REAL := 0.0;              (* Output from previous scan *)
END_VAR

(* 1. Initialization and Direct Bypass *)
IF InitCmd THEN
    CurrentValue := InitValue;
    PrevValue := InitValue;
    RampingUp := FALSE;
    RampingDown := FALSE;
    TargetReached := TRUE;
    DeltaRate := 0.0;
    RETURN;
ELSIF BypassRamp THEN
    CurrentValue := TargetValue;
    PrevValue := TargetValue;
    RampingUp := FALSE;
    RampingDown := FALSE;
    TargetReached := TRUE;
    DeltaRate := 0.0;
    RETURN;
END_IF;

(* 2. Step Limit Calculation *)
MaxUpStep := ABS(RampUpRate) * CycleTimeSec;
MaxDownStep := ABS(RampDownRate) * CycleTimeSec;
Difference := TargetValue - CurrentValue;

(* 3. Rate-Limiting Logic *)
IF ABS(Difference) <= Deadband THEN
    (* Target successfully reached within deadband *)
    CurrentValue := TargetValue;
    RampingUp := FALSE;
    RampingDown := FALSE;
    TargetReached := TRUE;
ELSIF Difference > 0.0 THEN
    (* Ascending toward TargetValue *)
    RampingUp := TRUE;
    RampingDown := FALSE;
    TargetReached := FALSE;

    IF Difference <= MaxUpStep THEN
        CurrentValue := TargetValue; (* Clamp to avoid overshoot *)
    ELSE
        CurrentValue := CurrentValue + MaxUpStep;
    END_IF;
ELSE
    (* Descending toward TargetValue *)
    RampingUp := FALSE;
    RampingDown := TRUE;
    TargetReached := FALSE;

    IF ABS(Difference) <= MaxDownStep THEN
        CurrentValue := TargetValue; (* Clamp to avoid overshoot *)
    ELSE
        CurrentValue := CurrentValue - MaxDownStep;
    END_IF;
END_IF;

(* 4. Velocity Calculation for Diagnostics *)
IF CycleTimeSec > 0.0001 THEN
    DeltaRate := (CurrentValue - PrevValue) / CycleTimeSec;
ELSE
    DeltaRate := 0.0;
END_IF;
PrevValue := CurrentValue;

END_FUNCTION_BLOCK

(* ---- turbine_ehc_overspeed_grid_sync.st ---- *)
(* ============================================================================
 * Title:       FB_TurbineEhcOverspeedGridSync
 * Description: Turbine Electro-Hydraulic Governor (EHC) Speed/Load Control,
 *              110% Mechanical/Electrical Overspeed Trip, Anti-Motoring Protection
 *              & Automatic Grid Synchronizer Interlock.
 * IEC 61131-3: Pure Structured Text (ST) Only. Ladder logic strictly rejected.
 * OCS Mapping:
 *   %R131: Turbine_Speed_RPM (INT: 0..4500 RPM, rated 3600 RPM)
 *   %R132: Generator_Active_Power_MW (INT: tenths of MW, e.g. 500 = 50.0 MW)
 *   %R133: Main_Stop_Valves_CV (INT: 0..100% position)
 *   %R134: Governor_Control_Valves_CV (INT: 0..100% position)
 *   %R135: Grid_Frequency_Hz (INT: hundredths of Hz, e.g. 6000 = 60.00 Hz)
 *   %R136: Phase_Angle_Error_Deg (INT: tenths of degree, e.g. 15 = 1.5 deg)
 *   %Q40:  ETS_Trip_Solenoid_Deenergize (BOOL: Emergency Trip System fail-safe)
 *   %Q41:  Generator_Breaker_Close_Permit (BOOL: Synch-check permit)
 *   %Q42:  EHC_Hydraulic_Pump_Run (BOOL: EHC fluid pump)
 *   %Q43:  Turbine_Turning_Gear_Engaged (BOOL: Rotor anti-sag turning gear)
 *   %M55:  Turbine_Overspeed_Trip_Latched (BOOL: Latched 110% overspeed trip)
 *   %M56:  Generator_Reverse_Power_Trip (BOOL: Latched reverse power trip)
 *   %M57:  Grid_Sync_Ready (BOOL: Speed, freq, phase angle in sync window)
 * ============================================================================ *)

FUNCTION_BLOCK FB_TurbineEhcOverspeedGridSync
VAR_INPUT
    Turbine_Speed_RPM : INT := 3600;            (* RPM (rated 3600) *)
    Generator_Active_Power_MW : INT := 500;     (* Tenths MW (500 = 50.0 MW) *)
    Grid_Frequency_Hz : INT := 6000;            (* Hundredths Hz (6000 = 60.00 Hz) *)
    Phase_Angle_Error_Deg : INT := 15;          (* Tenths deg (15 = 1.5 deg) *)
    EHC_Fluid_Pressure_OK : BOOL := TRUE;       (* Header pressure >= 1600 PSI *)
    Generator_Breaker_Closed : BOOL := TRUE;    (* Breaker auxiliary contact *)
    Master_Trip_Reset : BOOL := FALSE;          (* Operator trip reset PB *)
    Turning_Gear_Auto_Enable : BOOL := TRUE;    (* Auto turning gear permit *)
END_VAR

VAR_OUTPUT
    Main_Stop_Valves_CV : INT := 100;           (* 0..100% MSV position *)
    Governor_Control_Valves_CV : INT := 85;     (* 0..100% CV position *)
    ETS_Trip_Solenoid_Deenergize : BOOL := FALSE; (* Fail-safe trip *)
    Generator_Breaker_Close_Permit : BOOL := FALSE;
    EHC_Hydraulic_Pump_Run : BOOL := TRUE;
    Turbine_Turning_Gear_Engaged : BOOL := FALSE;
    Turbine_Overspeed_Trip_Latched : BOOL := FALSE;
    Generator_Reverse_Power_Trip : BOOL := FALSE;
    Grid_Sync_Ready : BOOL := FALSE;
END_VAR

VAR
    Overspeed_Setpoint_RPM : INT := 3960;       (* 110% of 3600 RPM *)
    Sync_Min_RPM : INT := 3595;
    Sync_Max_RPM : INT := 3605;
    Sync_Max_Phase_Deg : INT := 50;             (* 5.0 degrees *)
END_VAR

(* 0. Reset Latches *)
IF Master_Trip_Reset THEN
    Turbine_Overspeed_Trip_Latched := FALSE;
    Generator_Reverse_Power_Trip := FALSE;
    ETS_Trip_Solenoid_Deenergize := FALSE;
END_IF;

(* 1. Hydraulic Fluid Header Supervision *)
IF EHC_Fluid_Pressure_OK THEN
    EHC_Hydraulic_Pump_Run := TRUE;
ELSE
    EHC_Hydraulic_Pump_Run := FALSE;
    ETS_Trip_Solenoid_Deenergize := TRUE;
END_IF;

(* 2. Emergency Overspeed Protection (110% = 3960 RPM) *)
IF Turbine_Speed_RPM >= Overspeed_Setpoint_RPM THEN
    Turbine_Overspeed_Trip_Latched := TRUE;
    ETS_Trip_Solenoid_Deenergize := TRUE;
    Main_Stop_Valves_CV := 0;
    Governor_Control_Valves_CV := 0;
    Generator_Breaker_Close_Permit := FALSE;
    Grid_Sync_Ready := FALSE;
END_IF;

(* 3. Anti-Motoring / Reverse Power Protection (< -2.0 MW) *)
IF Generator_Breaker_Closed AND (Generator_Active_Power_MW <= -20) THEN
    Generator_Reverse_Power_Trip := TRUE;
    Generator_Breaker_Close_Permit := FALSE;
END_IF;

(* 4. Active Trip Enforcement *)
IF Turbine_Overspeed_Trip_Latched OR ETS_Trip_Solenoid_Deenergize THEN
    Main_Stop_Valves_CV := 0;
    Governor_Control_Valves_CV := 0;
    Generator_Breaker_Close_Permit := FALSE;
    Grid_Sync_Ready := FALSE;
END_IF;

(* 5. Automatic Grid Synchronizer Interlock *)
IF NOT Turbine_Overspeed_Trip_Latched AND NOT ETS_Trip_Solenoid_Deenergize THEN
    IF (Turbine_Speed_RPM >= Sync_Min_RPM) AND (Turbine_Speed_RPM <= Sync_Max_RPM) AND (Grid_Frequency_Hz >= 5990) AND (Grid_Frequency_Hz <= 6010) AND (Phase_Angle_Error_Deg <= Sync_Max_Phase_Deg) AND (Phase_Angle_Error_Deg >= -Sync_Max_Phase_Deg) THEN
        Grid_Sync_Ready := TRUE;
        Generator_Breaker_Close_Permit := TRUE;
    ELSE
        Grid_Sync_Ready := FALSE;
        IF NOT Generator_Breaker_Closed THEN
            Generator_Breaker_Close_Permit := FALSE;
        END_IF;
    END_IF;
END_IF;

(* 6. Cooldown Turning Gear Auto-Engagement (< 100 RPM) *)
IF Turning_Gear_Auto_Enable AND (Turbine_Speed_RPM < 100) AND (Main_Stop_Valves_CV = 0) THEN
    Turbine_Turning_Gear_Engaged := TRUE;
ELSE
    Turbine_Turning_Gear_Engaged := FALSE;
END_IF;

END_FUNCTION_BLOCK

(* ---- valve_actuator_controller.st ---- *)
(* ============================================================================
 * Title:       FB_ValveActuator
 * Description: Industrial Process Valve Actuator Controller with End-Position Watchdog.
 * Features:
 *   - Open and Close commanding with pulse or continuous solenoid output
 *   - Dual limit switch position feedback (Open and Closed end-stops)
 *   - Transit time watchdog timer detecting jammed or slow-stroking valves
 *   - Process safety interlock permissives inhibiting valve motion
 *   - Valve cycle counter and accumulated running transit time monitoring
 *   - Inconsistent limit switch fault detection (both open and closed active)
 * Language:    IEC 61131-3 Structured Text (Pure ST)
 * ============================================================================ *)

FUNCTION_BLOCK FB_ValveActuator
VAR_INPUT
    OpenCmd : BOOL := FALSE;              (* Request valve open command *)
    CloseCmd : BOOL := FALSE;             (* Request valve close command *)
    LimitOpen : BOOL := FALSE;            (* End-switch: Valve is fully open *)
    LimitClosed : BOOL := TRUE;           (* End-switch: Valve is fully closed *)
    InterlockOpen : BOOL := TRUE;         (* Safety permissive to permit opening (TRUE = OK) *)
    InterlockClose : BOOL := TRUE;        (* Safety permissive to permit closing (TRUE = OK) *)
    PulseMode : BOOL := FALSE;            (* TRUE = momentary solenoid pulse, FALSE = continuous *)
    PulseDurationSec : REAL := 2.0;       (* Pulse output hold duration (seconds) *)
    TransitTimeoutSec : REAL := 12.0;     (* Max permitted travel duration before travel fault *)
    ResetFault : BOOL := FALSE;           (* Push button to clear latched faults *)
    CycleTimeSec : REAL := 0.1;           (* Execution period of calling cyclic task (seconds) *)
END_VAR

VAR_OUTPUT
    SolOpen : BOOL := FALSE;              (* Physical digital output: Open solenoid / actuator *)
    SolClose : BOOL := FALSE;             (* Physical digital output: Close solenoid / actuator *)
    IsOpen : BOOL := FALSE;               (* Confirmed fully open state *)
    IsClosed : BOOL := TRUE;              (* Confirmed fully closed state *)
    IsTraveling : BOOL := FALSE;          (* Valve is currently in intermediate travel *)
    TravelFault : BOOL := FALSE;          (* Valve failed to reach target limit switch within timeout *)
    SwitchFault : BOOL := FALSE;          (* Sensor fault: Both open and closed limits are active simultaneously *)
    TotalCycles : DINT := 0;              (* Total full open-and-close cycles completed *)
    TransitTimeSec : REAL := 0.0;         (* Actual time taken during last complete stroke *)
END_VAR

VAR
    TargetOpen : BOOL := FALSE;           (* Desired position: TRUE = Open, FALSE = Closed *)
    TravelTimer : REAL := 0.0;            (* Elapsed stroke timer in seconds *)
    PulseTimer : REAL := 0.0;             (* Solenoid pulse energization timer *)
    PrevIsOpen : BOOL := FALSE;           (* Edge detection memory for cycle count *)
END_VAR

(* 1. Fault Reset *)
IF ResetFault THEN
    TravelFault := FALSE;
    SwitchFault := FALSE;
END_IF;

(* 2. Limit Switch Integrity Check *)
IF LimitOpen AND LimitClosed THEN
    SwitchFault := TRUE;
END_IF;

(* 3. Command Evaluation & Interlock Supervision *)
IF OpenCmd AND (NOT CloseCmd) THEN
    IF InterlockOpen AND (NOT TravelFault) AND (NOT SwitchFault) THEN
        TargetOpen := TRUE;
    END_IF;
ELSIF CloseCmd AND (NOT OpenCmd) THEN
    IF InterlockClose AND (NOT TravelFault) AND (NOT SwitchFault) THEN
        TargetOpen := FALSE;
    END_IF;
END_IF;

(* 4. Motion and Travel Timer Execution *)
IF TargetOpen THEN
    (* Commanding Open *)
    IF LimitOpen THEN
        (* Target reached *)
        SolOpen := FALSE;
        SolClose := FALSE;
        IsTraveling := FALSE;
        IF TravelTimer > 0.0 THEN
            TransitTimeSec := TravelTimer;
        END_IF;
        TravelTimer := 0.0;
        PulseTimer := 0.0;
    ELSE
        (* Currently in transit toward Open *)
        IsTraveling := TRUE;
        TravelTimer := TravelTimer + CycleTimeSec;

        IF TravelTimer >= TransitTimeoutSec THEN
            TravelFault := TRUE;
            SolOpen := FALSE;
            IsTraveling := FALSE;
        ELSE
            IF PulseMode THEN
                PulseTimer := PulseTimer + CycleTimeSec;
                SolOpen := PulseTimer <= PulseDurationSec;
            ELSE
                SolOpen := TRUE;
            END_IF;
            SolClose := FALSE;
        END_IF;
    END_IF;
ELSE
    (* Commanding Close *)
    IF LimitClosed THEN
        (* Target reached *)
        SolOpen := FALSE;
        SolClose := FALSE;
        IsTraveling := FALSE;
        IF TravelTimer > 0.0 THEN
            TransitTimeSec := TravelTimer;
        END_IF;
        TravelTimer := 0.0;
        PulseTimer := 0.0;
    ELSE
        (* Currently in transit toward Close *)
        IsTraveling := TRUE;
        TravelTimer := TravelTimer + CycleTimeSec;

        IF TravelTimer >= TransitTimeoutSec THEN
            TravelFault := TRUE;
            SolClose := FALSE;
            IsTraveling := FALSE;
        ELSE
            IF PulseMode THEN
                PulseTimer := PulseTimer + CycleTimeSec;
                SolClose := PulseTimer <= PulseDurationSec;
            ELSE
                SolClose := TRUE;
            END_IF;
            SolOpen := FALSE;
        END_IF;
    END_IF;
END_IF;

(* 5. Status Decoding *)
IsOpen := LimitOpen AND (NOT LimitClosed);
IsClosed := LimitClosed AND (NOT LimitOpen);

(* 6. Cycle Counter on confirmed full opening edge *)
IF IsOpen AND (NOT PrevIsOpen) THEN
    TotalCycles := TotalCycles + 1;
END_IF;
PrevIsOpen := IsOpen;

END_FUNCTION_BLOCK

(* ---- ccgt_hrsg_drum_level_duct_burner_control.st ---- *)
(* ============================================================================
   PROGRAM: CCGTHRSGDrumLevelDuctBurnerControl
   Standard: IEC 61131-3 Structured Text (ST Only)
   Target: Horner APG Cscape 10.2 / OCS Controller
   Description: Combined Cycle Gas Turbine (CCGT) Heat Recovery Steam Generator (HRSG)
                Three-Element Drum Level Control, Shrink/Swell Compensation, and
                Supplementary Firing Duct Burner Permissive Management.
                Pure Structured Text with zero ladder contacts/coils.
   ============================================================================ *)

PROGRAM CCGTHRSGDrumLevelDuctBurnerControl
VAR
    (* Analog Inputs (OCS %R Registers) *)
    DrumLevel_PV_mm            AT %R190 : REAL;    (* Drum level process variable (-500.0 to +500.0 mm) *)
    SteamFlow_Rate_kgs         AT %R191 : REAL;    (* Main high-pressure steam flow rate (0.0 to 120.0 kg/s) *)
    FeedwaterFlow_Rate_kgs     AT %R192 : REAL;    (* Boiler feedwater mass flow rate (0.0 to 120.0 kg/s) *)
    GT_ExhaustTemp_degC        AT %R193 : REAL;    (* Gas turbine exhaust gas temperature (400.0 to 650.0 C) *)
    DuctBurnerFiringDemand_pct AT %R194 : REAL;    (* Supplementary firing thermal demand (0.0 to 100.0%) *)
    FeedwaterValveOutput_pct   AT %R195 : REAL;    (* Feedwater control valve command (0.0 to 100.0%) *)
    DrumPressure_bar           AT %R196 : REAL;    (* Drum saturation operating pressure (0.0 to 120.0 bar) *)
    BlowdownFlow_Rate_kgs      AT %R197 : REAL;    (* Continuous/intermittent blowdown rate (0.0 to 10.0 kg/s) *)

    (* Digital Inputs (OCS %I Bits) *)
    GTRunPermissiveAux         AT %I36  : BOOL;    (* Gas turbine running permissive aux contact *)
    BoilerFeedPumpARunningAux  AT %I37  : BOOL;    (* Boiler feed pump A operational contact *)
    BoilerFeedPumpBRunningAux  AT %I38  : BOOL;    (* Boiler feed pump B operational contact *)
    DuctBurnerFlameDetected    AT %I39  : BOOL;    (* Duct burner scanner optical flame detected *)
    EmergencyTripResetPB       AT %I40  : BOOL;    (* Operator control room trip reset push-button *)

    (* Digital Outputs (OCS %Q Bits) *)
    FeedwaterControlAutoOnline AT %Q68  : BOOL;    (* Three-element feedwater control online *)
    DuctBurnerFuelGasBlockOpen AT %Q69  : BOOL;    (* Duct burner double block & bleed fuel valve open *)
    EmergencyBlowdownValveOpen AT %Q70  : BOOL;    (* High-level emergency blowdown dump valve open *)
    DrumProtectionCommonAlarm  AT %Q71  : BOOL;    (* HRSG drum protective annunciator common alarm *)

    (* Internal Flags (OCS %M Bits) *)
    ThreeElementModeActive     AT %M90  : BOOL;    (* True when steam and feedwater flow transmitters healthy *)
    DrumSwellShrinkActive      AT %M91  : BOOL;    (* Dynamic swell/shrink compensation bias applied *)
    HighDrumLevelWarning       AT %M92  : BOOL;    (* Level > +150.0 mm warning state *)
    LowDrumLevelWarning        AT %M93  : BOOL;    (* Level < -150.0 mm warning state *)
    LowLowDrumLevelTripLatched AT %M94  : BOOL;    (* Latched low-low level MFT trip (< -300.0 mm) *)
    HighHighDrumCarryoverTrip  AT %M95  : BOOL;    (* Latched high-high level carryover trip (> +350.0 mm) *)
    DuctBurnerPermissiveOK     AT %M96  : BOOL;    (* Supplementary firing interlocks satisfied *)
    BoilerMasterTripActive     AT %M97  : BOOL;    (* Common HRSG master trip state *)

    (* Setpoints & Design Limits *)
    DrumLevelSetpoint_mm       : REAL := 0.0;      (* Normal water level setpoint at centerline *)
    LowLowTripLimit_mm         : REAL := -300.0;   (* MFT low-low drum level trip point *)
    HighHighTripLimit_mm       : REAL := 350.0;    (* Steam turbine carryover high-high trip point *)
    MinGTExhaustTemp_degC      : REAL := 450.0;    (* Minimum GT exhaust temperature for duct firing *)
    MinFeedwaterFlow_kgs       : REAL := 5.0;      (* Minimum feedwater pump recirculation threshold *)

    (* Internal Process Calculation Registers *)
    LevelError_mm              : REAL := 0.0;
    FlowMismatch_kgs           : REAL := 0.0;
    TargetValvePos_pct         : REAL := 50.0;
END_VAR

(* ----------------------------------------------------------------------------
   Section 1: Operator Safety Reset Interlock
   ---------------------------------------------------------------------------- *)
IF EmergencyTripResetPB AND (BoilerFeedPumpARunningAux OR BoilerFeedPumpBRunningAux) THEN
    LowLowDrumLevelTripLatched := FALSE;
    HighHighDrumCarryoverTrip := FALSE;
    BoilerMasterTripActive := FALSE;
    DrumProtectionCommonAlarm := FALSE;
    EmergencyBlowdownValveOpen := FALSE;
END_IF;

(* ----------------------------------------------------------------------------
   Section 2: High-High Carryover and Low-Low Boil-Dry Protection
   ---------------------------------------------------------------------------- *)
IF DrumLevel_PV_mm < LowLowTripLimit_mm THEN
    LowLowDrumLevelTripLatched := TRUE;
    BoilerMasterTripActive := TRUE;
    DrumProtectionCommonAlarm := TRUE;
    DuctBurnerFuelGasBlockOpen := FALSE;
    FeedwaterControlAutoOnline := FALSE;
END_IF;

IF DrumLevel_PV_mm > HighHighTripLimit_mm THEN
    HighHighDrumCarryoverTrip := TRUE;
    BoilerMasterTripActive := TRUE;
    DrumProtectionCommonAlarm := TRUE;
    EmergencyBlowdownValveOpen := TRUE;
    DuctBurnerFuelGasBlockOpen := FALSE;
END_IF;

(* ----------------------------------------------------------------------------
   Section 3: Warning Threshold Monitoring
   ---------------------------------------------------------------------------- *)
HighDrumLevelWarning := (DrumLevel_PV_mm > 150.0) AND (NOT HighHighDrumCarryoverTrip);
LowDrumLevelWarning := (DrumLevel_PV_mm < -150.0) AND (NOT LowLowDrumLevelTripLatched);

(* ----------------------------------------------------------------------------
   Section 4: Supplementary Firing Duct Burner Permissive Logic
   Requires: GT running, exhaust temp > 450 C, at least 1 feed pump, no trips.
   ---------------------------------------------------------------------------- *)
DuctBurnerPermissiveOK := GTRunPermissiveAux
                          AND (GT_ExhaustTemp_degC >= MinGTExhaustTemp_degC)
                          AND (BoilerFeedPumpARunningAux OR BoilerFeedPumpBRunningAux)
                          AND (NOT BoilerMasterTripActive)
                          AND (DrumLevel_PV_mm > -200.0)
                          AND (DrumLevel_PV_mm < 200.0);

IF DuctBurnerPermissiveOK AND (DuctBurnerFiringDemand_pct > 5.0) THEN
    DuctBurnerFuelGasBlockOpen := TRUE;
ELSE
    DuctBurnerFuelGasBlockOpen := FALSE;
END_IF;

(* ----------------------------------------------------------------------------
   Section 5: Three-Element Drum Level & Dynamic Swell/Shrink Feedforward
   ---------------------------------------------------------------------------- *)
IF (NOT BoilerMasterTripActive) AND (BoilerFeedPumpARunningAux OR BoilerFeedPumpBRunningAux) THEN
    FeedwaterControlAutoOnline := TRUE;
    ThreeElementModeActive := TRUE;

    LevelError_mm := DrumLevelSetpoint_mm - DrumLevel_PV_mm;
    FlowMismatch_kgs := SteamFlow_Rate_kgs - FeedwaterFlow_Rate_kgs;

    (* Detect swell/shrink condition during rapid load changes *)
    IF (DuctBurnerFiringDemand_pct > 60.0) AND (SteamFlow_Rate_kgs > 75.0) THEN
        DrumSwellShrinkActive := TRUE;
    ELSE
        DrumSwellShrinkActive := FALSE;
    END_IF;

    (* Feedforward 3-element valve output calculation:
       Base position scales with steam flow, trimmed by level error and flow balance *)
    TargetValvePos_pct := (SteamFlow_Rate_kgs / 120.0) * 85.0 + (LevelError_mm * 0.05) + (FlowMismatch_kgs * 0.25);

    IF TargetValvePos_pct < 5.0 THEN
        FeedwaterValveOutput_pct := 5.0;
    ELSIF TargetValvePos_pct > 100.0 THEN
        FeedwaterValveOutput_pct := 100.0;
    ELSE
        FeedwaterValveOutput_pct := TargetValvePos_pct;
    END_IF;
ELSE
    FeedwaterControlAutoOnline := FALSE;
    ThreeElementModeActive := FALSE;
    FeedwaterValveOutput_pct := 0.0;
END_IF;

END_PROGRAM
